LIN {X 0,Y 433.476,Z 320.375,A -85,B 0,C 180,E1 -9833.026,E2 -9833.026} C_VEL
LIN {X 0,Y 436.058,Z 247.757,A -85,B 0,C 180,E1 -9834.679,E2 -9834.679} C_VEL
LIN {X 0,Y 438.537,Z 191.694,A -85,B 0,C 180,E1 -9836.045,E2 -9836.045} C_VEL
LIN {X 0,Y 435.909,Z 167.114,A -85,B 0,C 180,E1 -9837.032,E2 -9837.032} C_VEL
LIN {X 0,Y 432.859,Z 145.77,A -85,B 0,C 180,E1 -9838.059,E2 -9838.059} C_VEL
LIN {X 0,Y 426.886,Z 123.826,A -85,B 0,C 180,E1 -9841.119,E2 -9841.119} C_VEL
LIN {X 0,Y 425.305,Z 118.134,A -85,B 0,C 180,E1 -9841.978,E2 -9841.978} C_VEL
LIN {X 0,Y 425.294,Z 118.133,A -85,B 0,C 180,E1 -9845.337,E2 -9845.337} C_VEL
LIN {X 0,Y 425.279,Z 118.135,A -85,B 0,C 180,E1 -9848.901,E2 -9848.901} C_VEL
LIN {X 0,Y 425.255,Z 118.138,A -85,B 0,C 180,E1 -9852.656,E2 -9852.656} C_VEL
LIN {X 0,Y 425.284,Z 118.131,A -85,B 0,C 180,E1 -9855.283,E2 -9855.283} C_VEL
LIN {X 0,Y 425.247,Z 118.139,A -85,B 0,C 180,E1 -9858.618,E2 -9858.618} C_VEL
LIN {X 0,Y 425.279,Z 118.135,A -85,B 0,C 180,E1 -9861.1,E2 -9861.1} C_VEL
LIN {X 0,Y 425.294,Z 118.135,A -85,B 0,C 180,E1 -9864.664,E2 -9864.664} C_VEL
LIN {X 0,Y 425.262,Z 118.139,A -85,B 0,C 180,E1 -9868.073,E2 -9868.073} C_VEL
LIN {X 0,Y 425.304,Z 118.332,A -85,B 0,C 180,E1 -9870.341,E2 -9870.341} C_VEL
LIN {X 0,Y 427.302,Z 123.447,A -85,B 0,C 180,E1 -9871.42,E2 -9871.42} C_VEL
LIN {X 0,Y 432.761,Z 132.504,A -85,B 0,C 180,E1 -9872.386,E2 -9872.386} C_VEL
LIN {X 0,Y 437.753,Z 142.034,A -85,B 0,C 180,E1 -9873.231,E2 -9873.231} C_VEL
LIN {X 0,Y 440.603,Z 148.513,A -85,B 0,C 180,E1 -9873.713,E2 -9873.713} C_VEL
LIN {X 0,Y 436.849,Z 227.027,A -85,B 0,C 180,E1 -9875.622,E2 -9875.622} C_VEL
LIN {X 0,Y 434.621,Z 288.231,A -85,B 0,C 180,E1 -9877.039,E2 -9877.039} C_VEL
LIN {X 0,Y 433.965,Z 303.14,A -85,B 0,C 180,E1 -9877.553,E2 -9877.553} C_VEL
LIN {X 0,Y 433.141,Z 318.479,A -85,B 0,C 180,E1 -9878.276,E2 -9878.276} C_VEL
LIN {X 0,Y 432.336,Z 331.205,A -85,B 0,C 180,E1 -9879.046,E2 -9879.046} C_VEL
LIN {X 0,Y 431.344,Z 344.128,A -85,B 0,C 180,E1 -9879.992,E2 -9879.992} C_VEL
LIN {X 0,Y 430.278,Z 357.22,A -85,B 0,C 180,E1 -9881.159,E2 -9881.159} C_VEL
LIN {X 0,Y 429.205,Z 368.572,A -85,B 0,C 180,E1 -9882.367,E2 -9882.367} C_VEL
LIN {X 0,Y 428.183,Z 379.818,A -85,B 0,C 180,E1 -9883.798,E2 -9883.798} C_VEL
LIN {X 0,Y 427.387,Z 389.291,A -85,B 0,C 180,E1 -9885.234,E2 -9885.234} C_VEL
LIN {X 0,Y 426.432,Z 398.569,A -85,B 0,C 180,E1 -9886.903,E2 -9886.903} C_VEL
LIN {X 0,Y 425.775,Z 406.243,A -85,B 0,C 180,E1 -9888.576,E2 -9888.576} C_VEL
LIN {X 0,Y 425.268,Z 413.343,A -85,B 0,C 180,E1 -9890.488,E2 -9890.488} C_VEL
LIN {X 0,Y 424.809,Z 418.9,A -85,B 0,C 180,E1 -9892.395,E2 -9892.395} C_VEL
LIN {X 0,Y 424.497,Z 423.037,A -85,B 0,C 180,E1 -9894.299,E2 -9894.299} C_VEL
LIN {X 0,Y 424.444,Z 425.857,A -85,B 0,C 180,E1 -9896.203,E2 -9896.203} C_VEL
LIN {X 0,Y 424.285,Z 427.454,A -85,B 0,C 180,E1 -9898.102,E2 -9898.102} C_VEL
LIN {X 0,Y 424.198,Z 427.83,A -85,B 0,C 180,E1 -9900,E2 -9900} C_VEL
LIN {X 0,Y 424.232,Z 426.986,A -85,B 0,C 180,E1 -9901.899,E2 -9901.899} C_VEL
LIN {X 0,Y 424.347,Z 424.903,A -85,B 0,C 180,E1 -9903.799,E2 -9903.799} C_VEL
LIN {X 0,Y 424.456,Z 421.542,A -85,B 0,C 180,E1 -9905.702,E2 -9905.702} C_VEL
LIN {X 0,Y 424.638,Z 416.847,A -85,B 0,C 180,E1 -9907.609,E2 -9907.609} C_VEL
LIN {X 0,Y 424.941,Z 410.703,A -85,B 0,C 180,E1 -9909.52,E2 -9909.52} C_VEL
LIN {X 0,Y 425.467,Z 402.93,A -85,B 0,C 180,E1 -9911.433,E2 -9911.433} C_VEL
LIN {X 0,Y 425.898,Z 394.118,A -85,B 0,C 180,E1 -9913.196,E2 -9913.196} C_VEL
LIN {X 0,Y 426.684,Z 384.46,A -85,B 0,C 180,E1 -9914.792,E2 -9914.792} C_VEL
LIN {X 0,Y 427.452,Z 374.109,A -85,B 0,C 180,E1 -9916.231,E2 -9916.231} C_VEL
LIN {X 0,Y 428.404,Z 361.628,A -85,B 0,C 180,E1 -9917.678,E2 -9917.678} C_VEL
LIN {X 0,Y 429.284,Z 349.36,A -85,B 0,C 180,E1 -9918.865,E2 -9918.865} C_VEL
LIN {X 0,Y 430.123,Z 335.923,A -85,B 0,C 180,E1 -9919.944,E2 -9919.944} C_VEL
LIN {X 0,Y 431.021,Z 321.131,A -85,B 0,C 180,E1 -9920.897,E2 -9920.897} C_VEL
LIN {X 0,Y 431.726,Z 306.43,A -85,B 0,C 180,E1 -9921.642,E2 -9921.642} C_VEL
LIN {X 0,Y 432.318,Z 290.546,A -85,B 0,C 180,E1 -9922.239,E2 -9922.239} C_VEL
LIN {X 0,Y 432.751,Z 273.967,A -85,B 0,C 180,E1 -9922.656,E2 -9922.656} C_VEL
LIN {X 0,Y 435.763,Z 148.938,A -85,B 0,C 180,E1 -9925.144,E2 -9925.144} C_VEL
LIN {X 0,Y 435.826,Z 144.558,A -85,B 0,C 180,E1 -9925.236,E2 -9925.236} C_VEL
LIN {X 0,Y 427.552,Z 123.717,A -85,B 0,C 180,E1 -9926.145,E2 -9926.145} C_VEL
LIN {X 0,Y 425.381,Z 118.566,A -85,B 0,C 180,E1 -9926.383,E2 -9926.383} C_VEL
LIN {X 0,Y 425.309,Z 118.131,A -85,B 0,C 180,E1 -9926.44,E2 -9926.44} C_VEL
LIN {X 0,Y 425.285,Z 118.138,A -85,B 0,C 180,E1 -9929.72,E2 -9929.72} C_VEL
LIN {X 0,Y 425.271,Z 118.136,A -85,B 0,C 180,E1 -9933.049,E2 -9933.049} C_VEL
LIN {X 0,Y 425.282,Z 118.135,A -85,B 0,C 180,E1 -9935.928,E2 -9935.928} C_VEL
LIN {X 0,Y 425.264,Z 118.137,A -85,B 0,C 180,E1 -9939.038,E2 -9939.038} C_VEL
LIN {X 0,Y 425.259,Z 118.135,A -85,B 0,C 180,E1 -9942.656,E2 -9942.656} C_VEL
LIN {X 0,Y 425.287,Z 118.121,A -85,B 0,C 180,E1 -9945.283,E2 -9945.283} C_VEL
LIN {X 0,Y 425.251,Z 118.129,A -85,B 0,C 180,E1 -9948.619,E2 -9948.619} C_VEL
LIN {X 0,Y 425.286,Z 118.138,A -85,B 0,C 180,E1 -9951.1,E2 -9951.1} C_VEL
LIN {X 0,Y 425.297,Z 118.117,A -85,B 0,C 180,E1 -9954.664,E2 -9954.664} C_VEL
LIN {X 0,Y 425.263,Z 118.135,A -85,B 0,C 180,E1 -9958.073,E2 -9958.073} C_VEL
LIN {X 0,Y 425.307,Z 118.126,A -85,B 0,C 180,E1 -9961.366,E2 -9961.366} C_VEL
LIN {X 0,Y 425.263,Z 118.137,A -85,B 0,C 180,E1 -9964.553,E2 -9964.553} C_VEL
LIN {X 0,Y 425.294,Z 118.131,A -85,B 0,C 180,E1 -9967.73,E2 -9967.73} C_VEL
LIN {X 0,Y 425.363,Z 118.121,A -85,B 0,C 180,E1 -9970.704,E2 -9970.704} C_VEL
LIN {X 0,Y 425.326,Z 118.123,A -85,B 0,C 180,E1 -9973.686,E2 -9973.686} C_VEL
LIN {X 0,Y 425.397,Z 118.118,A -85,B 0,C 180,E1 -9977.097,E2 -9977.097} C_VEL
LIN {X 0,Y 425.391,Z 118.118,A -85,B 0,C 180,E1 -9977.809,E2 -9977.809} C_VEL
LIN {X 0,Y 424.671,Z 118.212,A -85,B 0,C 180,E1 -9978.599,E2 -9978.599} C_VEL
LIN {X 0,Y 421.798,Z 118.565,A -85,B 0,C 180,E1 -9979.883,E2 -9979.883} C_VEL
LIN {X 0,Y 419.433,Z 118.863,A -85,B 0,C 180,E1 -9980.92,E2 -9980.92} C_VEL
LIN {X 0,Y 418.468,Z 118.982,A -85,B 0,C 180,E1 -9981.721,E2 -9981.721} C_VEL
LIN {X 0,Y 418.414,Z 118.988,A -85,B 0,C 180,E1 -9981.992,E2 -9981.992} C_VEL
LIN {X 0,Y 418.469,Z 118.985,A -85,B 0,C 180,E1 -9984.217,E2 -9984.217} C_VEL
LIN {X 0,Y 418.285,Z 119.156,A -85,B 0,C 180,E1 -9986.177,E2 -9986.177} C_VEL
LIN {X 0,Y 420.692,Z 127.345,A -85,B 0,C 180,E1 -9987.606,E2 -9987.606} C_VEL
LIN {X 0,Y 424.262,Z 143.272,A -85,B 0,C 180,E1 -9990.245,E2 -9990.245} C_VEL
LIN {X 0,Y 427.065,Z 154.574,A -85,B 0,C 180,E1 -9990.638,E2 -9990.638} C_VEL
LIN {X 0,Y 430.401,Z 170.837,A -85,B 0,C 180,E1 -9991.151,E2 -9991.151} C_VEL
LIN {X 0,Y 427.922,Z 309.723,A -85,B 0,C 180,E1 -9993.56,E2 -9993.56} C_VEL
LIN {X 0,Y 427.342,Z 325.024,A -85,B 0,C 180,E1 -9994.008,E2 -9994.008} C_VEL
LIN {X 0,Y 426.606,Z 339.301,A -85,B 0,C 180,E1 -9994.606,E2 -9994.606} C_VEL
LIN {X 0,Y 425.719,Z 352.541,A -85,B 0,C 180,E1 -9995.328,E2 -9995.328} C_VEL
LIN {X 0,Y 424.65,Z 366.851,A -85,B 0,C 180,E1 -9996.323,E2 -9996.323} C_VEL
LIN {X 0,Y 423.516,Z 379.354,A -85,B 0,C 180,E1 -9997.389,E2 -9997.389} C_VEL
LIN {X 0,Y 422.318,Z 392.27,A -85,B 0,C 180,E1 -9998.734,E2 -9998.734} C_VEL
LIN {X 0,Y 421.206,Z 403.348,A -85,B 0,C 180,E1 -10000.118,E2 -10000.118} C_VEL
LIN {X 0,Y 420.207,Z 413.193,A -85,B 0,C 180,E1 -10001.578,E2 -10001.578} C_VEL
LIN {X 0,Y 419.231,Z 423.087,A -85,B 0,C 180,E1 -10003.344,E2 -10003.344} C_VEL
LIN {X 0,Y 418.471,Z 431.173,A -85,B 0,C 180,E1 -10005.089,E2 -10005.089} C_VEL
LIN {X 0,Y 417.884,Z 438.749,A -85,B 0,C 180,E1 -10007.117,E2 -10007.117} C_VEL
LIN {X 0,Y 417.436,Z 444.47,A -85,B 0,C 180,E1 -10009.055,E2 -10009.055} C_VEL
LIN {X 0,Y 417.228,Z 448.297,A -85,B 0,C 180,E1 -10010.716,E2 -10010.716} C_VEL
LIN {X 0,Y 416.957,Z 451.799,A -85,B 0,C 180,E1 -10012.81,E2 -10012.81} C_VEL
LIN {X 0,Y 416.84,Z 453.914,A -85,B 0,C 180,E1 -10014.93,E2 -10014.93} C_VEL
LIN {X 0,Y 416.81,Z 454.647,A -85,B 0,C 180,E1 -10017.082,E2 -10017.082} C_VEL
LIN {X 0,Y 416.88,Z 453.936,A -85,B 0,C 180,E1 -10019.268,E2 -10019.268} C_VEL
LIN {X 0,Y 416.959,Z 452.622,A -85,B 0,C 180,E1 -10020.725,E2 -10020.725} C_VEL
LIN {X 0,Y 417.123,Z 449.953,A -85,B 0,C 180,E1 -10022.626,E2 -10022.626} C_VEL
LIN {X 0,Y 417.374,Z 446.422,A -85,B 0,C 180,E1 -10024.401,E2 -10024.401} C_VEL
LIN {X 0,Y 417.655,Z 441.894,A -85,B 0,C 180,E1 -10026.127,E2 -10026.127} C_VEL
LIN {X 0,Y 418.184,Z 435.407,A -85,B 0,C 180,E1 -10028.086,E2 -10028.086} C_VEL
LIN {X 0,Y 418.9,Z 427.843,A -85,B 0,C 180,E1 -10029.921,E2 -10029.921} C_VEL
LIN {X 0,Y 419.836,Z 418.621,A -85,B 0,C 180,E1 -10031.754,E2 -10031.754} C_VEL
LIN {X 0,Y 420.792,Z 409.737,A -85,B 0,C 180,E1 -10033.218,E2 -10033.218} C_VEL
LIN {X 0,Y 421.901,Z 398.872,A -85,B 0,C 180,E1 -10034.733,E2 -10034.733} C_VEL
LIN {X 0,Y 423.054,Z 387.69,A -85,B 0,C 180,E1 -10036.035,E2 -10036.035} C_VEL
LIN {X 0,Y 424.244,Z 375.52,A -85,B 0,C 180,E1 -10037.218,E2 -10037.218} C_VEL
LIN {X 0,Y 425.412,Z 362.05,A -85,B 0,C 180,E1 -10038.296,E2 -10038.296} C_VEL
LIN {X 0,Y 426.457,Z 348.268,A -85,B 0,C 180,E1 -10039.182,E2 -10039.182} C_VEL
LIN {X 0,Y 427.423,Z 333.071,A -85,B 0,C 180,E1 -10039.937,E2 -10039.937} C_VEL
LIN {X 0,Y 428.11,Z 318.612,A -85,B 0,C 180,E1 -10040.459,E2 -10040.459} C_VEL
LIN {X 0,Y 428.609,Z 302.995,A -85,B 0,C 180,E1 -10040.831,E2 -10040.831} C_VEL
LIN {X 0,Y 431.166,Z 166.127,A -85,B 0,C 180,E1 -10043.203,E2 -10043.203} C_VEL
LIN {X 0,Y 427.935,Z 148.87,A -85,B 0,C 180,E1 -10043.755,E2 -10043.755} C_VEL
LIN {X 0,Y 424.959,Z 141.623,A -85,B 0,C 180,E1 -10044.132,E2 -10044.132} C_VEL
LIN {X 0,Y 421.22,Z 128.241,A -85,B 0,C 180,E1 -10046.017,E2 -10046.017} C_VEL
LIN {X 0,Y 418.253,Z 119.013,A -85,B 0,C 180,E1 -10047.386,E2 -10047.386} C_VEL
LIN {X 0,Y 418.271,Z 119.005,A -85,B 0,C 180,E1 -10050.895,E2 -10050.895} C_VEL
LIN {X 0,Y 418.343,Z 119.17,A -85,B 0,C 180,E1 -10053.285,E2 -10053.285} C_VEL
LIN {X 0,Y 420.465,Z 124.425,A -85,B 0,C 180,E1 -10053.527,E2 -10053.527} C_VEL
LIN {X 0,Y 428.257,Z 143.1,A -85,B 0,C 180,E1 -10054.384,E2 -10054.384} C_VEL
LIN {X 0,Y 429.352,Z 145.894,A -85,B 0,C 180,E1 -10054.505,E2 -10054.505} C_VEL
LIN {X 0,Y 425.813,Z 284.514,A -85,B 0,C 180,E1 -10057.37,E2 -10057.37} C_VEL
LIN {X 0,Y 425.291,Z 300.109,A -85,B 0,C 180,E1 -10057.884,E2 -10057.884} C_VEL
LIN {X 0,Y 424.58,Z 315.42,A -85,B 0,C 180,E1 -10058.585,E2 -10058.585} C_VEL
LIN {X 0,Y 423.681,Z 330.521,A -85,B 0,C 180,E1 -10059.487,E2 -10059.487} C_VEL
LIN {X 0,Y 422.828,Z 343.594,A -85,B 0,C 180,E1 -10060.457,E2 -10060.457} C_VEL
LIN {X 0,Y 421.904,Z 356.853,A -85,B 0,C 180,E1 -10061.655,E2 -10061.655} C_VEL
LIN {X 0,Y 420.946,Z 369.299,A -85,B 0,C 180,E1 -10063.011,E2 -10063.011} C_VEL
LIN {X 0,Y 420.094,Z 380.508,A -85,B 0,C 180,E1 -10064.474,E2 -10064.474} C_VEL
LIN {X 0,Y 419.355,Z 389.987,A -85,B 0,C 180,E1 -10065.936,E2 -10065.936} C_VEL
LIN {X 0,Y 418.741,Z 399.242,A -85,B 0,C 180,E1 -10067.643,E2 -10067.643} C_VEL
LIN {X 0,Y 418.126,Z 406.928,A -85,B 0,C 180,E1 -10069.345,E2 -10069.345} C_VEL
LIN {X 0,Y 417.739,Z 414.027,A -85,B 0,C 180,E1 -10071.291,E2 -10071.291} C_VEL
LIN {X 0,Y 417.441,Z 419.577,A -85,B 0,C 180,E1 -10073.232,E2 -10073.232} C_VEL
LIN {X 0,Y 417.253,Z 423.717,A -85,B 0,C 180,E1 -10075.169,E2 -10075.169} C_VEL
LIN {X 0,Y 417.274,Z 426.53,A -85,B 0,C 180,E1 -10077.103,E2 -10077.103} C_VEL
LIN {X 0,Y 417.116,Z 428.105,A -85,B 0,C 180,E1 -10079.034,E2 -10079.034} C_VEL
LIN {X 0,Y 417.159,Z 428.456,A -85,B 0,C 180,E1 -10080.965,E2 -10080.965} C_VEL
LIN {X 0,Y 417.307,Z 427.591,A -85,B 0,C 180,E1 -10082.896,E2 -10082.896} C_VEL
LIN {X 0,Y 417.35,Z 425.512,A -85,B 0,C 180,E1 -10084.83,E2 -10084.83} C_VEL
LIN {X 0,Y 417.706,Z 421.785,A -85,B 0,C 180,E1 -10086.933,E2 -10086.933} C_VEL
LIN {X 0,Y 418.018,Z 417.459,A -85,B 0,C 180,E1 -10088.703,E2 -10088.703} C_VEL
LIN {X 0,Y 418.538,Z 411.293,A -85,B 0,C 180,E1 -10090.644,E2 -10090.644} C_VEL
LIN {X 0,Y 419.232,Z 403.488,A -85,B 0,C 180,E1 -10092.587,E2 -10092.587} C_VEL
LIN {X 0,Y 420.006,Z 395.644,A -85,B 0,C 180,E1 -10094.189,E2 -10094.189} C_VEL
LIN {X 0,Y 420.973,Z 386.577,A -85,B 0,C 180,E1 -10095.741,E2 -10095.741} C_VEL
LIN {X 0,Y 421.96,Z 376.468,A -85,B 0,C 180,E1 -10097.195,E2 -10097.195} C_VEL
LIN {X 0,Y 423.082,Z 364.868,A -85,B 0,C 180,E1 -10098.601,E2 -10098.601} C_VEL
LIN {X 0,Y 424.377,Z 351.134,A -85,B 0,C 180,E1 -10099.972,E2 -10099.972} C_VEL
LIN {X 0,Y 425.556,Z 337.924,A -85,B 0,C 180,E1 -10101.051,E2 -10101.051} C_VEL
LIN {X 0,Y 426.562,Z 323.478,A -85,B 0,C 180,E1 -10102.013,E2 -10102.013} C_VEL
LIN {X 0,Y 427.571,Z 308.227,A -85,B 0,C 180,E1 -10102.802,E2 -10102.802} C_VEL
LIN {X 0,Y 428.387,Z 292.392,A -85,B 0,C 180,E1 -10103.411,E2 -10103.411} C_VEL
LIN {X 0,Y 429.03,Z 274.518,A -85,B 0,C 180,E1 -10103.886,E2 -10103.886} C_VEL
LIN {X 0,Y 432.057,Z 206.122,A -85,B 0,C 180,E1 -10105.535,E2 -10105.535} C_VEL
LIN {X 0,Y 435.05,Z 152.54,A -85,B 0,C 180,E1 -10106.899,E2 -10106.899} C_VEL
LIN {X 0,Y 429.528,Z 141.704,A -85,B 0,C 180,E1 -10107.869,E2 -10107.869} C_VEL
LIN {X 0,Y 423.452,Z 131.573,A -85,B 0,C 180,E1 -10108.995,E2 -10108.995} C_VEL
LIN {X 0,Y 421.069,Z 127.829,A -85,B 0,C 180,E1 -10109.498,E2 -10109.498} C_VEL
LIN {X 0,Y 419.163,Z 121.743,A -85,B 0,C 180,E1 -10111.88,E2 -10111.88} C_VEL
LIN {X 0,Y 418.224,Z 119.016,A -85,B 0,C 180,E1 -10113.214,E2 -10113.214} C_VEL
LIN {X 0,Y 418.243,Z 119.013,A -85,B 0,C 180,E1 -10116.237,E2 -10116.237} C_VEL
LIN {X 0,Y 418.199,Z 119.02,A -85,B 0,C 180,E1 -10119.688,E2 -10119.688} C_VEL
LIN {X 0,Y 418.207,Z 119.018,A -85,B 0,C 180,E1 -10122.318,E2 -10122.318} C_VEL
LIN {X 0,Y 418.234,Z 119.014,A -85,B 0,C 180,E1 -10125.108,E2 -10125.108} C_VEL
LIN {X 0,Y 418.218,Z 119.017,A -85,B 0,C 180,E1 -10127.764,E2 -10127.764} C_VEL
LIN {X 0,Y 418.264,Z 119.189,A -85,B 0,C 180,E1 -10131.251,E2 -10131.251} C_VEL
LIN {X 0,Y 420.236,Z 124.674,A -85,B 0,C 180,E1 -10133.393,E2 -10133.393} C_VEL
LIN {X 0,Y 422.812,Z 132.475,A -85,B 0,C 180,E1 -10135.857,E2 -10135.857} C_VEL
LIN {X 0,Y 425.058,Z 140.837,A -85,B 0,C 180,E1 -10138.056,E2 -10138.056} C_VEL
LIN {X 0,Y 427.012,Z 150.076,A -85,B 0,C 180,E1 -10140.141,E2 -10140.141} C_VEL
LIN {X 0,Y 426.311,Z 155.998,A -85,B 0,C 180,E1 -10141.195,E2 -10141.195} C_VEL
LIN {X 0,Y 429.906,Z 173.135,A -85,B 0,C 180,E1 -10142.192,E2 -10142.192} C_VEL
LIN {X 0,Y 432.21,Z 187.065,A -85,B 0,C 180,E1 -10142.874,E2 -10142.874} C_VEL
LIN {X 0,Y 433.425,Z 198.784,A -85,B 0,C 180,E1 -10143.353,E2 -10143.353} C_VEL
LIN {X 0,Y 429.495,Z 281.182,A -85,B 0,C 180,E1 -10145.37,E2 -10145.37} C_VEL
LIN {X 0,Y 427.704,Z 328.281,A -85,B 0,C 180,E1 -10146.485,E2 -10146.485} C_VEL
LIN {X 0,Y 426.584,Z 344.904,A -85,B 0,C 180,E1 -10147.062,E2 -10147.062} C_VEL
LIN {X 0,Y 425.045,Z 368.196,A -85,B 0,C 180,E1 -10148.155,E2 -10148.155} C_VEL
LIN {X 0,Y 424.013,Z 381.982,A -85,B 0,C 180,E1 -10148.996,E2 -10148.996} C_VEL
LIN {X 0,Y 423.04,Z 394.637,A -85,B 0,C 180,E1 -10149.962,E2 -10149.962} C_VEL
LIN {X 0,Y 421.807,Z 407.625,A -85,B 0,C 180,E1 -10151.166,E2 -10151.166} C_VEL
LIN {X 0,Y 420.765,Z 419.459,A -85,B 0,C 180,E1 -10152.503,E2 -10152.503} C_VEL
LIN {X 0,Y 419.746,Z 430.266,A -85,B 0,C 180,E1 -10153.962,E2 -10153.962} C_VEL
LIN {X 0,Y 418.815,Z 440.763,A -85,B 0,C 180,E1 -10155.669,E2 -10155.669} C_VEL
LIN {X 0,Y 418.115,Z 449.456,A -85,B 0,C 180,E1 -10157.378,E2 -10157.378} C_VEL
LIN {X 0,Y 417.766,Z 455.753,A -85,B 0,C 180,E1 -10158.845,E2 -10158.845} C_VEL
LIN {X 0,Y 417.329,Z 462.608,A -85,B 0,C 180,E1 -10160.794,E2 -10160.794} C_VEL
LIN {X 0,Y 417.183,Z 467.962,A -85,B 0,C 180,E1 -10162.741,E2 -10162.741} C_VEL
LIN {X 0,Y 417.089,Z 471.027,A -85,B 0,C 180,E1 -10164.197,E2 -10164.197} C_VEL
LIN {X 0,Y 417.015,Z 474.038,A -85,B 0,C 180,E1 -10166.135,E2 -10166.135} C_VEL
LIN {X 0,Y 417.107,Z 475.831,A -85,B 0,C 180,E1 -10168.069,E2 -10168.069} C_VEL
LIN {X 0,Y 417.008,Z 476.43,A -85,B 0,C 180,E1 -10170,E2 -10170} C_VEL
LIN {X 0,Y 417.105,Z 475.816,A -85,B 0,C 180,E1 -10171.931,E2 -10171.931} C_VEL
LIN {X 0,Y 417.022,Z 473.988,A -85,B 0,C 180,E1 -10173.865,E2 -10173.865} C_VEL
LIN {X 0,Y 417.103,Z 470.93,A -85,B 0,C 180,E1 -10175.802,E2 -10175.802} C_VEL
LIN {X 0,Y 417.213,Z 466.566,A -85,B 0,C 180,E1 -10177.745,E2 -10177.745} C_VEL
LIN {X 0,Y 417.373,Z 460.79,A -85,B 0,C 180,E1 -10179.694,E2 -10179.694} C_VEL
LIN {X 0,Y 417.826,Z 453.441,A -85,B 0,C 180,E1 -10181.645,E2 -10181.645} C_VEL
LIN {X 0,Y 418.352,Z 445.454,A -85,B 0,C 180,E1 -10183.367,E2 -10183.367} C_VEL
LIN {X 0,Y 419.132,Z 435.942,A -85,B 0,C 180,E1 -10185.064,E2 -10185.064} C_VEL
LIN {X 0,Y 420.01,Z 426.133,A -85,B 0,C 180,E1 -10186.527,E2 -10186.527} C_VEL
LIN {X 0,Y 420.865,Z 415.606,A -85,B 0,C 180,E1 -10187.855,E2 -10187.855} C_VEL
LIN {X 0,Y 421.863,Z 403.993,A -85,B 0,C 180,E1 -10189.083,E2 -10189.083} C_VEL
LIN {X 0,Y 422.961,Z 391.607,A -85,B 0,C 180,E1 -10190.169,E2 -10190.169} C_VEL
LIN {X 0,Y 423.984,Z 378.111,A -85,B 0,C 180,E1 -10191.133,E2 -10191.133} C_VEL
LIN {X 0,Y 425.004,Z 363.864,A -85,B 0,C 180,E1 -10191.929,E2 -10191.929} C_VEL
LIN {X 0,Y 425.699,Z 349.61,A -85,B 0,C 180,E1 -10192.54,E2 -10192.54} C_VEL
LIN {X 0,Y 426.927,Z 326.53,A -85,B 0,C 180,E1 -10193.303,E2 -10193.303} C_VEL
LIN {X 0,Y 430.632,Z 235.57,A -85,B 0,C 180,E1 -10195.466,E2 -10195.466} C_VEL
LIN {X 0,Y 432.676,Z 192.835,A -85,B 0,C 180,E1 -10196.555,E2 -10196.555} C_VEL
LIN {X 0,Y 430.315,Z 169.02,A -85,B 0,C 180,E1 -10197.549,E2 -10197.549} C_VEL
LIN {X 0,Y 427.476,Z 148.909,A -85,B 0,C 180,E1 -10198.546,E2 -10198.546} C_VEL
LIN {X 0,Y 423.411,Z 137.794,A -85,B 0,C 180,E1 -10199.581,E2 -10199.581} C_VEL
LIN {X 0,Y 418.279,Z 119.007,A -85,B 0,C 180,E1 -10202.311,E2 -10202.311} C_VEL
LIN {X 0,Y 418.249,Z 119.013,A -85,B 0,C 180,E1 -10204.842,E2 -10204.842} C_VEL
LIN {X 0,Y 418.237,Z 119.012,A -85,B 0,C 180,E1 -10208.444,E2 -10208.444} C_VEL
LIN {X 0,Y 418.218,Z 119.012,A -85,B 0,C 180,E1 -10212.236,E2 -10212.236} C_VEL
LIN {X 0,Y 418.234,Z 119.01,A -85,B 0,C 180,E1 -10215.109,E2 -10215.109} C_VEL
LIN {X 0,Y 418.218,Z 119.012,A -85,B 0,C 180,E1 -10217.764,E2 -10217.764} C_VEL
LIN {X 0,Y 418.237,Z 119.014,A -85,B 0,C 180,E1 -10221.557,E2 -10221.557} C_VEL
LIN {X 0,Y 418.25,Z 119.012,A -85,B 0,C 180,E1 -10225.158,E2 -10225.158} C_VEL
LIN {X 0,Y 418.243,Z 119.013,A -85,B 0,C 180,E1 -10227.472,E2 -10227.472} C_VEL
LIN {X 0,Y 418.275,Z 119.133,A -85,B 0,C 180,E1 -10229.366,E2 -10229.366} C_VEL
LIN {X 0,Y 418.771,Z 120.997,A -85,B 0,C 180,E1 -10229.77,E2 -10229.77} C_VEL
LIN {X 0,Y 420.148,Z 123.987,A -85,B 0,C 180,E1 -10230.487,E2 -10230.487} C_VEL
LIN {X 0,Y 426.123,Z 133.617,A -85,B 0,C 180,E1 -10231.643,E2 -10231.643} C_VEL
LIN {X 0,Y 430.993,Z 142.386,A -85,B 0,C 180,E1 -10232.52,E2 -10232.52} C_VEL
LIN {X 0,Y 434.88,Z 150.985,A -85,B 0,C 180,E1 -10233.217,E2 -10233.217} C_VEL
LIN {X 0,Y 430.518,Z 234.6,A -85,B 0,C 180,E1 -10235.304,E2 -10235.304} C_VEL
LIN {X 0,Y 428.335,Z 289.381,A -85,B 0,C 180,E1 -10236.618,E2 -10236.618} C_VEL
LIN {X 0,Y 427.588,Z 305.204,A -85,B 0,C 180,E1 -10237.19,E2 -10237.19} C_VEL
LIN {X 0,Y 426.693,Z 320.173,A -85,B 0,C 180,E1 -10237.93,E2 -10237.93} C_VEL
LIN {X 0,Y 425.713,Z 334.367,A -85,B 0,C 180,E1 -10238.831,E2 -10238.831} C_VEL
LIN {X 0,Y 424.548,Z 348.176,A -85,B 0,C 180,E1 -10239.91,E2 -10239.91} C_VEL
LIN {X 0,Y 423.39,Z 360.836,A -85,B 0,C 180,E1 -10241.114,E2 -10241.114} C_VEL
LIN {X 0,Y 422.308,Z 371.547,A -85,B 0,C 180,E1 -10242.319,E2 -10242.319} C_VEL
LIN {X 0,Y 421.288,Z 382.377,A -85,B 0,C 180,E1 -10243.774,E2 -10243.774} C_VEL
LIN {X 0,Y 420.398,Z 391.524,A -85,B 0,C 180,E1 -10245.23,E2 -10245.23} C_VEL
LIN {X 0,Y 419.431,Z 400.498,A -85,B 0,C 180,E1 -10246.926,E2 -10246.926} C_VEL
LIN {X 0,Y 418.837,Z 406.906,A -85,B 0,C 180,E1 -10248.384,E2 -10248.384} C_VEL
LIN {X 0,Y 418.279,Z 413.962,A -85,B 0,C 180,E1 -10250.327,E2 -10250.327} C_VEL
LIN {X 0,Y 417.792,Z 419.473,A -85,B 0,C 180,E1 -10252.266,E2 -10252.266} C_VEL
LIN {X 0,Y 417.455,Z 423.565,A -85,B 0,C 180,E1 -10254.203,E2 -10254.203} C_VEL
LIN {X 0,Y 417.384,Z 426.346,A -85,B 0,C 180,E1 -10256.138,E2 -10256.138} C_VEL
LIN {X 0,Y 417.208,Z 427.896,A -85,B 0,C 180,E1 -10258.07,E2 -10258.07} C_VEL
LIN {X 0,Y 417.112,Z 428.222,A -85,B 0,C 180,E1 -10260,E2 -10260} C_VEL
LIN {X 0,Y 417.157,Z 427.324,A -85,B 0,C 180,E1 -10261.931,E2 -10261.931} C_VEL
LIN {X 0,Y 417.252,Z 425.193,A -85,B 0,C 180,E1 -10263.863,E2 -10263.863} C_VEL
LIN {X 0,Y 417.383,Z 421.774,A -85,B 0,C 180,E1 -10265.799,E2 -10265.799} C_VEL
LIN {X 0,Y 417.574,Z 417.004,A -85,B 0,C 180,E1 -10267.738,E2 -10267.738} C_VEL
LIN {X 0,Y 417.882,Z 410.774,A -85,B 0,C 180,E1 -10269.682,E2 -10269.682} C_VEL
LIN {X 0,Y 418.355,Z 403.949,A -85,B 0,C 180,E1 -10271.385,E2 -10271.385} C_VEL
LIN {X 0,Y 418.738,Z 396.907,A -85,B 0,C 180,E1 -10272.858,E2 -10272.858} C_VEL
LIN {X 0,Y 419.503,Z 387.256,A -85,B 0,C 180,E1 -10274.555,E2 -10274.555} C_VEL
LIN {X 0,Y 420.289,Z 377.336,A -85,B 0,C 180,E1 -10276.017,E2 -10276.017} C_VEL
LIN {X 0,Y 421.228,Z 365.533,A -85,B 0,C 180,E1 -10277.477,E2 -10277.477} C_VEL
LIN {X 0,Y 422.124,Z 352.523,A -85,B 0,C 180,E1 -10278.819,E2 -10278.819} C_VEL
LIN {X 0,Y 423.049,Z 339.692,A -85,B 0,C 180,E1 -10279.911,E2 -10279.911} C_VEL
LIN {X 0,Y 423.936,Z 325.787,A -85,B 0,C 180,E1 -10280.881,E2 -10280.881} C_VEL
LIN {X 0,Y 424.746,Z 310.546,A -85,B 0,C 180,E1 -10281.724,E2 -10281.724} C_VEL
LIN {X 0,Y 425.373,Z 295.193,A -85,B 0,C 180,E1 -10282.366,E2 -10282.366} C_VEL
LIN {X 0,Y 425.868,Z 279.661,A -85,B 0,C 180,E1 -10282.819,E2 -10282.819} C_VEL
LIN {X 0,Y 429.149,Z 149.841,A -85,B 0,C 180,E1 -10285.474,E2 -10285.474} C_VEL
LIN {X 0,Y 429.007,Z 145.736,A -85,B 0,C 180,E1 -10285.573,E2 -10285.573} C_VEL
LIN {X 0,Y 421.571,Z 127.049,A -85,B 0,C 180,E1 -10286.402,E2 -10286.402} C_VEL
LIN {X 0,Y 418.336,Z 119.6,A -85,B 0,C 180,E1 -10286.757,E2 -10286.757} C_VEL
LIN {X 0,Y 418.245,Z 119.012,A -85,B 0,C 180,E1 -10286.792,E2 -10286.792} C_VEL
LIN {X 0,Y 418.243,Z 119.012,A -85,B 0,C 180,E1 -10290.273,E2 -10290.273} C_VEL
LIN {X 0,Y 418.234,Z 119.015,A -85,B 0,C 180,E1 -10293.679,E2 -10293.679} C_VEL
LIN {X 0,Y 418.24,Z 119.013,A -85,B 0,C 180,E1 -10297.225,E2 -10297.225} C_VEL
LIN {X 0,Y 418.209,Z 119.015,A -85,B 0,C 180,E1 -10300.867,E2 -10300.867} C_VEL
LIN {X 0,Y 418.205,Z 119.012,A -85,B 0,C 180,E1 -10303.729,E2 -10303.729} C_VEL
LIN {X 0,Y 418.201,Z 118.995,A -85,B 0,C 180,E1 -10306.448,E2 -10306.448} C_VEL
LIN {X 0,Y 418.212,Z 119.011,A -85,B 0,C 180,E1 -10309.133,E2 -10309.133} C_VEL
LIN {X 0,Y 418.241,Z 119.007,A -85,B 0,C 180,E1 -10312.776,E2 -10312.776} C_VEL
LIN {X 0,Y 418.235,Z 119.007,A -85,B 0,C 180,E1 -10316.322,E2 -10316.322} C_VEL
LIN {X 0,Y 418.241,Z 119.002,A -85,B 0,C 180,E1 -10319.728,E2 -10319.728} C_VEL
LIN {X 0,Y 418.224,Z 119.017,A -85,B 0,C 180,E1 -10323.017,E2 -10323.017} C_VEL
LIN {X 0,Y 418.258,Z 118.999,A -85,B 0,C 180,E1 -10326.217,E2 -10326.217} C_VEL
LIN {X 0,Y 418.25,Z 119.005,A -85,B 0,C 180,E1 -10329.337,E2 -10329.337} C_VEL
LIN {X 0,Y 418.259,Z 119.013,A -85,B 0,C 180,E1 -10332.395,E2 -10332.395} C_VEL
LIN {X 0,Y 418.279,Z 119.007,A -85,B 0,C 180,E1 -10335.402,E2 -10335.402} C_VEL
LIN {X 0,Y 418.316,Z 119.007,A -85,B 0,C 180,E1 -10338.369,E2 -10338.369} C_VEL
LIN {X 0,Y 418.414,Z 118.988,A -85,B 0,C 180,E1 -10341.992,E2 -10341.992} C_VEL
LIN {X 0,Y 417.781,Z 119.072,A -85,B 0,C 180,E1 -10342.527,E2 -10342.527} C_VEL
LIN {X 0,Y 414.954,Z 119.422,A -85,B 0,C 180,E1 -10343.364,E2 -10343.364} C_VEL
LIN {X 0,Y 412.046,Z 119.786,A -85,B 0,C 180,E1 -10344.211,E2 -10344.211} C_VEL
LIN {X 0,Y 411.318,Z 119.874,A -85,B 0,C 180,E1 -10344.76,E2 -10344.76} C_VEL
LIN {X 0,Y 411.243,Z 120.098,A -85,B 0,C 180,E1 -10345.774,E2 -10345.774} C_VEL
LIN {X 0,Y 414.2,Z 130.215,A -85,B 0,C 180,E1 -10347.569,E2 -10347.569} C_VEL
LIN {X 0,Y 417.199,Z 143.468,A -85,B 0,C 180,E1 -10349.779,E2 -10349.779} C_VEL
LIN {X 0,Y 419.11,Z 149.054,A -85,B 0,C 180,E1 -10350.015,E2 -10350.015} C_VEL
LIN {X 0,Y 423.908,Z 171.508,A -85,B 0,C 180,E1 -10350.754,E2 -10350.754} C_VEL
LIN {X 0,Y 421.374,Z 309.968,A -85,B 0,C 180,E1 -10353.197,E2 -10353.197} C_VEL
LIN {X 0,Y 420.768,Z 325.254,A -85,B 0,C 180,E1 -10353.651,E2 -10353.651} C_VEL
LIN {X 0,Y 419.996,Z 339.529,A -85,B 0,C 180,E1 -10354.258,E2 -10354.258} C_VEL
LIN {X 0,Y 418.992,Z 353.707,A -85,B 0,C 180,E1 -10355.052,E2 -10355.052} C_VEL
LIN {X 0,Y 418.005,Z 366.432,A -85,B 0,C 180,E1 -10355.948,E2 -10355.948} C_VEL
LIN {X 0,Y 416.7,Z 380.204,A -85,B 0,C 180,E1 -10357.145,E2 -10357.145} C_VEL
LIN {X 0,Y 415.474,Z 393.004,A -85,B 0,C 180,E1 -10358.512,E2 -10358.512} C_VEL
LIN {X 0,Y 414.396,Z 402.934,A -85,B 0,C 180,E1 -10359.764,E2 -10359.764} C_VEL
LIN {X 0,Y 413.338,Z 413.023,A -85,B 0,C 180,E1 -10361.276,E2 -10361.276} C_VEL
LIN {X 0,Y 412.443,Z 421.575,A -85,B 0,C 180,E1 -10362.798,E2 -10362.798} C_VEL
LIN {X 0,Y 411.591,Z 430.017,A -85,B 0,C 180,E1 -10364.588,E2 -10364.588} C_VEL
LIN {X 0,Y 411.009,Z 436.636,A -85,B 0,C 180,E1 -10366.289,E2 -10366.289} C_VEL
LIN {X 0,Y 410.581,Z 441.966,A -85,B 0,C 180,E1 -10367.945,E2 -10367.945} C_VEL
LIN {X 0,Y 410.224,Z 447.252,A -85,B 0,C 180,E1 -10370.038,E2 -10370.038} C_VEL
LIN {X 0,Y 409.936,Z 451.206,A -85,B 0,C 180,E1 -10372.212,E2 -10372.212} C_VEL
LIN {X 0,Y 409.796,Z 453.62,A -85,B 0,C 180,E1 -10374.305,E2 -10374.305} C_VEL
LIN {X 0,Y 409.712,Z 454.737,A -85,B 0,C 180,E1 -10376.487,E2 -10376.487} C_VEL
LIN {X 0,Y 409.754,Z 454.434,A -85,B 0,C 180,E1 -10378.702,E2 -10378.702} C_VEL
LIN {X 0,Y 409.878,Z 452.637,A -85,B 0,C 180,E1 -10380.957,E2 -10380.957} C_VEL
LIN {X 0,Y 410.056,Z 449.892,A -85,B 0,C 180,E1 -10382.878,E2 -10382.878} C_VEL
LIN {X 0,Y 410.347,Z 446.214,A -85,B 0,C 180,E1 -10384.704,E2 -10384.704} C_VEL
LIN {X 0,Y 410.773,Z 440.618,A -85,B 0,C 180,E1 -10386.786,E2 -10386.786} C_VEL
LIN {X 0,Y 411.344,Z 434.323,A -85,B 0,C 180,E1 -10388.629,E2 -10388.629} C_VEL
LIN {X 0,Y 412.037,Z 426.919,A -85,B 0,C 180,E1 -10390.403,E2 -10390.403} C_VEL
LIN {X 0,Y 413.06,Z 417.626,A -85,B 0,C 180,E1 -10392.227,E2 -10392.227} C_VEL
LIN {X 0,Y 414.172,Z 408.105,A -85,B 0,C 180,E1 -10393.784,E2 -10393.784} C_VEL
LIN {X 0,Y 415.339,Z 397.121,A -85,B 0,C 180,E1 -10395.291,E2 -10395.291} C_VEL
LIN {X 0,Y 416.636,Z 384.993,A -85,B 0,C 180,E1 -10396.673,E2 -10396.673} C_VEL
LIN {X 0,Y 417.972,Z 371.929,A -85,B 0,C 180,E1 -10397.897,E2 -10397.897} C_VEL
LIN {X 0,Y 419.132,Z 358.932,A -85,B 0,C 180,E1 -10398.896,E2 -10398.896} C_VEL
LIN {X 0,Y 420.225,Z 344.402,A -85,B 0,C 180,E1 -10399.785,E2 -10399.785} C_VEL
LIN {X 0,Y 421.163,Z 329.225,A -85,B 0,C 180,E1 -10400.488,E2 -10400.488} C_VEL
LIN {X 0,Y 421.827,Z 315.103,A -85,B 0,C 180,E1 -10400.958,E2 -10400.958} C_VEL
LIN {X 0,Y 422.254,Z 297.455,A -85,B 0,C 180,E1 -10401.331,E2 -10401.331} C_VEL
LIN {X 0,Y 424.783,Z 166.685,A -85,B 0,C 180,E1 -10403.636,E2 -10403.636} C_VEL
LIN {X 0,Y 421.932,Z 151.429,A -85,B 0,C 180,E1 -10404.138,E2 -10404.138} C_VEL
LIN {X 0,Y 417.911,Z 141.886,A -85,B 0,C 180,E1 -10404.647,E2 -10404.647} C_VEL
LIN {X 0,Y 414.136,Z 128.828,A -85,B 0,C 180,E1 -10406.529,E2 -10406.529} C_VEL
LIN {X 0,Y 411.174,Z 119.893,A -85,B 0,C 180,E1 -10407.859,E2 -10407.859} C_VEL
LIN {X 0,Y 411.221,Z 119.887,A -85,B 0,C 180,E1 -10411.41,E2 -10411.41} C_VEL
LIN {X 0,Y 411.277,Z 119.882,A -85,B 0,C 180,E1 -10412.881,E2 -10412.881} C_VEL
LIN {X 0,Y 412.965,Z 124.424,A -85,B 0,C 180,E1 -10413.096,E2 -10413.096} C_VEL
LIN {X 0,Y 420.673,Z 142.445,A -85,B 0,C 180,E1 -10413.953,E2 -10413.953} C_VEL
LIN {X 0,Y 422.777,Z 148.152,A -85,B 0,C 180,E1 -10414.199,E2 -10414.199} C_VEL
LIN {X 0,Y 419.045,Z 284.518,A -85,B 0,C 180,E1 -10417.082,E2 -10417.082} C_VEL
LIN {X 0,Y 418.509,Z 300.304,A -85,B 0,C 180,E1 -10417.61,E2 -10417.61} C_VEL
LIN {X 0,Y 417.811,Z 314.865,A -85,B 0,C 180,E1 -10418.28,E2 -10418.28} C_VEL
LIN {X 0,Y 416.942,Z 329.33,A -85,B 0,C 180,E1 -10419.14,E2 -10419.14} C_VEL
LIN {X 0,Y 416.036,Z 342.687,A -85,B 0,C 180,E1 -10420.125,E2 -10420.125} C_VEL
LIN {X 0,Y 415.144,Z 355.124,A -85,B 0,C 180,E1 -10421.237,E2 -10421.237} C_VEL
LIN {X 0,Y 414.197,Z 367.798,A -85,B 0,C 180,E1 -10422.599,E2 -10422.599} C_VEL
LIN {X 0,Y 413.158,Z 380.173,A -85,B 0,C 180,E1 -10424.206,E2 -10424.206} C_VEL
LIN {X 0,Y 412.389,Z 389.783,A -85,B 0,C 180,E1 -10425.693,E2 -10425.693} C_VEL
LIN {X 0,Y 411.737,Z 399.159,A -85,B 0,C 180,E1 -10427.43,E2 -10427.43} C_VEL
LIN {X 0,Y 411.097,Z 406.925,A -85,B 0,C 180,E1 -10429.16,E2 -10429.16} C_VEL
LIN {X 0,Y 410.698,Z 414.136,A -85,B 0,C 180,E1 -10431.14,E2 -10431.14} C_VEL
LIN {X 0,Y 410.381,Z 419.766,A -85,B 0,C 180,E1 -10433.115,E2 -10433.115} C_VEL
LIN {X 0,Y 410.189,Z 423.967,A -85,B 0,C 180,E1 -10435.085,E2 -10435.085} C_VEL
LIN {X 0,Y 410.208,Z 426.842,A -85,B 0,C 180,E1 -10437.053,E2 -10437.053} C_VEL
LIN {X 0,Y 410.035,Z 428.482,A -85,B 0,C 180,E1 -10439.018,E2 -10439.018} C_VEL
LIN {X 0,Y 410.077,Z 428.892,A -85,B 0,C 180,E1 -10440.982,E2 -10440.982} C_VEL
LIN {X 0,Y 410.243,Z 428.078,A -85,B 0,C 180,E1 -10442.946,E2 -10442.946} C_VEL
LIN {X 0,Y 410.343,Z 427.214,A -85,B 0,C 180,E1 -10443.928,E2 -10443.928} C_VEL
LIN {X 0,Y 410.428,Z 424.561,A -85,B 0,C 180,E1 -10445.897,E2 -10445.897} C_VEL
LIN {X 0,Y 410.767,Z 420.595,A -85,B 0,C 180,E1 -10447.867,E2 -10447.867} C_VEL
LIN {X 0,Y 411.337,Z 415.23,A -85,B 0,C 180,E1 -10449.837,E2 -10449.837} C_VEL
LIN {X 0,Y 411.942,Z 408.33,A -85,B 0,C 180,E1 -10451.813,E2 -10451.813} C_VEL
LIN {X 0,Y 412.682,Z 400.898,A -85,B 0,C 180,E1 -10453.54,E2 -10453.54} C_VEL
LIN {X 0,Y 413.754,Z 391.859,A -85,B 0,C 180,E1 -10455.265,E2 -10455.265} C_VEL
LIN {X 0,Y 414.866,Z 380.956,A -85,B 0,C 180,E1 -10456.991,E2 -10456.991} C_VEL
LIN {X 0,Y 416.066,Z 369.74,A -85,B 0,C 180,E1 -10458.464,E2 -10458.464} C_VEL
LIN {X 0,Y 417.341,Z 357.436,A -85,B 0,C 180,E1 -10459.81,E2 -10459.81} C_VEL
LIN {X 0,Y 418.468,Z 345.502,A -85,B 0,C 180,E1 -10460.909,E2 -10460.909} C_VEL
LIN {X 0,Y 419.717,Z 330.912,A -85,B 0,C 180,E1 -10462.003,E2 -10462.003} C_VEL
LIN {X 0,Y 420.734,Z 317.464,A -85,B 0,C 180,E1 -10462.818,E2 -10462.818} C_VEL
LIN {X 0,Y 421.711,Z 302.301,A -85,B 0,C 180,E1 -10463.529,E2 -10463.529} C_VEL
LIN {X 0,Y 422.426,Z 287.203,A -85,B 0,C 180,E1 -10464.054,E2 -10464.054} C_VEL
LIN {X 0,Y 425.929,Z 212.161,A -85,B 0,C 180,E1 -10465.929,E2 -10465.929} C_VEL
LIN {X 0,Y 429.311,Z 154.969,A -85,B 0,C 180,E1 -10467.44,E2 -10467.44} C_VEL
LIN {X 0,Y 424.311,Z 145.12,A -85,B 0,C 180,E1 -10468.377,E2 -10468.377} C_VEL
LIN {X 0,Y 418.912,Z 136.263,A -85,B 0,C 180,E1 -10469.424,E2 -10469.424} C_VEL
LIN {X 0,Y 416.225,Z 132.205,A -85,B 0,C 180,E1 -10469.985,E2 -10469.985} C_VEL
LIN {X 0,Y 414.228,Z 128.978,A -85,B 0,C 180,E1 -10470.455,E2 -10470.455} C_VEL
LIN {X 0,Y 412.259,Z 123.067,A -85,B 0,C 180,E1 -10473.06,E2 -10473.06} C_VEL
LIN {X 0,Y 411.206,Z 119.89,A -85,B 0,C 180,E1 -10474.877,E2 -10474.877} C_VEL
LIN {X 0,Y 411.194,Z 119.891,A -85,B 0,C 180,E1 -10478.166,E2 -10478.166} C_VEL
LIN {X 0,Y 411.159,Z 119.895,A -85,B 0,C 180,E1 -10481.807,E2 -10481.807} C_VEL
LIN {X 0,Y 411.173,Z 119.894,A -85,B 0,C 180,E1 -10485.509,E2 -10485.509} C_VEL
LIN {X 0,Y 411.146,Z 119.899,A -85,B 0,C 180,E1 -10488.774,E2 -10488.774} C_VEL
LIN {X 0,Y 411.155,Z 120.03,A -85,B 0,C 180,E1 -10489.602,E2 -10489.602} C_VEL
LIN {X 0,Y 412.615,Z 124.153,A -85,B 0,C 180,E1 -10491.583,E2 -10491.583} C_VEL
LIN {X 0,Y 414.865,Z 130.353,A -85,B 0,C 180,E1 -10493.971,E2 -10493.971} C_VEL
LIN {X 0,Y 417.139,Z 137.573,A -85,B 0,C 180,E1 -10496.221,E2 -10496.221} C_VEL
LIN {X 0,Y 419.256,Z 145.957,A -85,B 0,C 180,E1 -10498.41,E2 -10498.41} C_VEL
LIN {X 0,Y 420.518,Z 152.505,A -85,B 0,C 180,E1 -10499.909,E2 -10499.909} C_VEL
LIN {X 0,Y 420.282,Z 155.554,A -85,B 0,C 180,E1 -10500.434,E2 -10500.434} C_VEL
LIN {X 0,Y 423.58,Z 170.608,A -85,B 0,C 180,E1 -10501.391,E2 -10501.391} C_VEL
LIN {X 0,Y 426.324,Z 186.91,A -85,B 0,C 180,E1 -10502.262,E2 -10502.262} C_VEL
LIN {X 0,Y 427.663,Z 199.684,A -85,B 0,C 180,E1 -10502.818,E2 -10502.818} C_VEL
LIN {X 0,Y 423.4,Z 281.775,A -85,B 0,C 180,E1 -10504.893,E2 -10504.893} C_VEL
LIN {X 0,Y 421.421,Z 328.643,A -85,B 0,C 180,E1 -10506.047,E2 -10506.047} C_VEL
LIN {X 0,Y 420.182,Z 345.469,A -85,B 0,C 180,E1 -10506.656,E2 -10506.656} C_VEL
LIN {X 0,Y 418.513,Z 367.645,A -85,B 0,C 180,E1 -10507.76,E2 -10507.76} C_VEL
LIN {X 0,Y 417.371,Z 381.99,A -85,B 0,C 180,E1 -10508.645,E2 -10508.645} C_VEL
LIN {X 0,Y 416.342,Z 394.587,A -85,B 0,C 180,E1 -10509.625,E2 -10509.625} C_VEL
LIN {X 0,Y 415.065,Z 407.548,A -85,B 0,C 180,E1 -10510.849,E2 -10510.849} C_VEL
LIN {X 0,Y 413.95,Z 419.363,A -85,B 0,C 180,E1 -10512.206,E2 -10512.206} C_VEL
LIN {X 0,Y 412.842,Z 430.154,A -85,B 0,C 180,E1 -10513.687,E2 -10513.687} C_VEL
LIN {X 0,Y 411.877,Z 440.638,A -85,B 0,C 180,E1 -10515.423,E2 -10515.423} C_VEL
LIN {X 0,Y 411.112,Z 449.32,A -85,B 0,C 180,E1 -10517.16,E2 -10517.16} C_VEL
LIN {X 0,Y 410.73,Z 455.608,A -85,B 0,C 180,E1 -10518.651,E2 -10518.651} C_VEL
LIN {X 0,Y 410.251,Z 462.449,A -85,B 0,C 180,E1 -10520.634,E2 -10520.634} C_VEL
LIN {X 0,Y 410.112,Z 467.794,A -85,B 0,C 180,E1 -10522.616,E2 -10522.616} C_VEL
LIN {X 0,Y 409.996,Z 470.854,A -85,B 0,C 180,E1 -10524.097,E2 -10524.097} C_VEL
LIN {X 0,Y 409.931,Z 473.861,A -85,B 0,C 180,E1 -10526.068,E2 -10526.068} C_VEL
LIN {X 0,Y 410.031,Z 475.649,A -85,B 0,C 180,E1 -10528.035,E2 -10528.035} C_VEL
LIN {X 0,Y 409.93,Z 476.244,A -85,B 0,C 180,E1 -10530,E2 -10530} C_VEL
LIN {X 0,Y 410.03,Z 475.626,A -85,B 0,C 180,E1 -10531.965,E2 -10531.965} C_VEL
LIN {X 0,Y 409.937,Z 473.791,A -85,B 0,C 180,E1 -10533.932,E2 -10533.932} C_VEL
LIN {X 0,Y 410.013,Z 470.725,A -85,B 0,C 180,E1 -10535.903,E2 -10535.903} C_VEL
LIN {X 0,Y 410.132,Z 466.353,A -85,B 0,C 180,E1 -10537.879,E2 -10537.879} C_VEL
LIN {X 0,Y 410.306,Z 460.567,A -85,B 0,C 180,E1 -10539.863,E2 -10539.863} C_VEL
LIN {X 0,Y 410.757,Z 454.223,A -85,B 0,C 180,E1 -10541.598,E2 -10541.598} C_VEL
LIN {X 0,Y 411.261,Z 446.75,A -85,B 0,C 180,E1 -10543.288,E2 -10543.288} C_VEL
LIN {X 0,Y 412.054,Z 437.162,A -85,B 0,C 180,E1 -10545.076,E2 -10545.076} C_VEL
LIN {X 0,Y 412.951,Z 427.623,A -85,B 0,C 180,E1 -10546.563,E2 -10546.563} C_VEL
LIN {X 0,Y 413.948,Z 416.188,A -85,B 0,C 180,E1 -10548.054,E2 -10548.054} C_VEL
LIN {X 0,Y 414.986,Z 404.919,A -85,B 0,C 180,E1 -10549.284,E2 -10549.284} C_VEL
LIN {X 0,Y 416.106,Z 392.725,A -85,B 0,C 180,E1 -10550.387,E2 -10550.387} C_VEL
LIN {X 0,Y 417.176,Z 379.522,A -85,B 0,C 180,E1 -10551.365,E2 -10551.365} C_VEL
LIN {X 0,Y 418.22,Z 365.909,A -85,B 0,C 180,E1 -10552.163,E2 -10552.163} C_VEL
LIN {X 0,Y 418.976,Z 351.328,A -85,B 0,C 180,E1 -10552.824,E2 -10552.824} C_VEL
LIN {X 0,Y 420.213,Z 333.683,A -85,B 0,C 180,E1 -10553.535,E2 -10553.535} C_VEL
LIN {X 0,Y 421.101,Z 316.689,A -85,B 0,C 180,E1 -10554.005,E2 -10554.005} C_VEL
LIN {X 0,Y 424.275,Z 244.479,A -85,B 0,C 180,E1 -10555.77,E2 -10555.77} C_VEL
LIN {X 0,Y 426.922,Z 193.664,A -85,B 0,C 180,E1 -10557.101,E2 -10557.101} C_VEL
LIN {X 0,Y 424.748,Z 170.445,A -85,B 0,C 180,E1 -10558.115,E2 -10558.115} C_VEL
LIN {X 0,Y 422.272,Z 152.134,A -85,B 0,C 180,E1 -10559.06,E2 -10559.06} C_VEL
LIN {X 0,Y 418.745,Z 142.594,A -85,B 0,C 180,E1 -10559.935,E2 -10559.935} C_VEL
LIN {X 0,Y 412.63,Z 124.982,A -85,B 0,C 180,E1 -10561.961,E2 -10561.961} C_VEL
LIN {X 0,Y 411.222,Z 119.886,A -85,B 0,C 180,E1 -10562.662,E2 -10562.662} C_VEL
LIN {X 0,Y 411.177,Z 119.891,A -85,B 0,C 180,E1 -10565.531,E2 -10565.531} C_VEL
LIN {X 0,Y 411.178,Z 119.893,A -85,B 0,C 180,E1 -10569.229,E2 -10569.229} C_VEL
LIN {X 0,Y 411.165,Z 119.893,A -85,B 0,C 180,E1 -10572.694,E2 -10572.694} C_VEL
LIN {X 0,Y 411.163,Z 119.889,A -85,B 0,C 180,E1 -10575.882,E2 -10575.882} C_VEL
LIN {X 0,Y 411.157,Z 119.893,A -85,B 0,C 180,E1 -10579.493,E2 -10579.493} C_VEL
LIN {X 0,Y 411.185,Z 119.893,A -85,B 0,C 180,E1 -10582.026,E2 -10582.026} C_VEL
LIN {X 0,Y 411.202,Z 119.89,A -85,B 0,C 180,E1 -10585.123,E2 -10585.123} C_VEL
LIN {X 0,Y 411.184,Z 120.032,A -85,B 0,C 180,E1 -10588.256,E2 -10588.256} C_VEL
LIN {X 0,Y 412.044,Z 122.478,A -85,B 0,C 180,E1 -10588.871,E2 -10588.871} C_VEL
LIN {X 0,Y 413.47,Z 125.421,A -85,B 0,C 180,E1 -10589.552,E2 -10589.552} C_VEL
LIN {X 0,Y 417.515,Z 131.455,A -85,B 0,C 180,E1 -10590.421,E2 -10590.421} C_VEL
LIN {X 0,Y 421.958,Z 138.843,A -85,B 0,C 180,E1 -10591.31,E2 -10591.31} C_VEL
LIN {X 0,Y 427.048,Z 148.462,A -85,B 0,C 180,E1 -10592.277,E2 -10592.277} C_VEL
LIN {X 0,Y 429.202,Z 153.375,A -85,B 0,C 180,E1 -10592.691,E2 -10592.691} C_VEL
LIN {X 0,Y 424.385,Z 237.716,A -85,B 0,C 180,E1 -10594.857,E2 -10594.857} C_VEL
LIN {X 0,Y 422.175,Z 289.509,A -85,B 0,C 180,E1 -10596.146,E2 -10596.146} C_VEL
LIN {X 0,Y 421.303,Z 306.222,A -85,B 0,C 180,E1 -10596.764,E2 -10596.764} C_VEL
LIN {X 0,Y 420.355,Z 320.975,A -85,B 0,C 180,E1 -10597.515,E2 -10597.515} C_VEL
LIN {X 0,Y 419.371,Z 334.215,A -85,B 0,C 180,E1 -10598.366,E2 -10598.366} C_VEL
LIN {X 0,Y 418.157,Z 348.086,A -85,B 0,C 180,E1 -10599.461,E2 -10599.461} C_VEL
LIN {X 0,Y 416.94,Z 360.573,A -85,B 0,C 180,E1 -10600.656,E2 -10600.656} C_VEL
LIN {X 0,Y 415.838,Z 370.534,A -85,B 0,C 180,E1 -10601.78,E2 -10601.78} C_VEL
LIN {X 0,Y 414.649,Z 381.594,A -85,B 0,C 180,E1 -10603.254,E2 -10603.254} C_VEL
LIN {X 0,Y 413.586,Z 392.351,A -85,B 0,C 180,E1 -10604.981,E2 -10604.981} C_VEL
LIN {X 0,Y 412.549,Z 401.26,A -85,B 0,C 180,E1 -10606.704,E2 -10606.704} C_VEL
LIN {X 0,Y 411.897,Z 407.61,A -85,B 0,C 180,E1 -10608.185,E2 -10608.185} C_VEL
LIN {X 0,Y 411.281,Z 414.615,A -85,B 0,C 180,E1 -10610.161,E2 -10610.161} C_VEL
LIN {X 0,Y 410.766,Z 420.07,A -85,B 0,C 180,E1 -10612.133,E2 -10612.133} C_VEL
LIN {X 0,Y 410.416,Z 424.116,A -85,B 0,C 180,E1 -10614.103,E2 -10614.103} C_VEL
LIN {X 0,Y 410.326,Z 426.846,A -85,B 0,C 180,E1 -10616.072,E2 -10616.072} C_VEL
LIN {X 0,Y 410.133,Z 428.344,A -85,B 0,C 180,E1 -10618.036,E2 -10618.036} C_VEL
LIN {X 0,Y 410.029,Z 428.616,A -85,B 0,C 180,E1 -10620,E2 -10620} C_VEL
LIN {X 0,Y 410.085,Z 427.656,A -85,B 0,C 180,E1 -10621.965,E2 -10621.965} C_VEL
LIN {X 0,Y 410.194,Z 426.713,A -85,B 0,C 180,E1 -10622.947,E2 -10622.947} C_VEL
LIN {X 0,Y 410.173,Z 423.891,A -85,B 0,C 180,E1 -10624.915,E2 -10624.915} C_VEL
LIN {X 0,Y 410.394,Z 419.738,A -85,B 0,C 180,E1 -10626.885,E2 -10626.885} C_VEL
LIN {X 0,Y 410.676,Z 414.17,A -85,B 0,C 180,E1 -10628.86,E2 -10628.86} C_VEL
LIN {X 0,Y 411.062,Z 407.024,A -85,B 0,C 180,E1 -10630.84,E2 -10630.84} C_VEL
LIN {X 0,Y 411.66,Z 399.326,A -85,B 0,C 180,E1 -10632.573,E2 -10632.573} C_VEL
LIN {X 0,Y 412.201,Z 391.427,A -85,B 0,C 180,E1 -10634.062,E2 -10634.062} C_VEL
LIN {X 0,Y 412.923,Z 382.157,A -85,B 0,C 180,E1 -10635.55,E2 -10635.55} C_VEL
LIN {X 0,Y 413.816,Z 371.197,A -85,B 0,C 180,E1 -10637.036,E2 -10637.036} C_VEL
LIN {X 0,Y 414.726,Z 359.399,A -85,B 0,C 180,E1 -10638.38,E2 -10638.38} C_VEL
LIN {X 0,Y 415.76,Z 346.206,A -85,B 0,C 180,E1 -10639.632,E2 -10639.632} C_VEL
LIN {X 0,Y 416.569,Z 333.626,A -85,B 0,C 180,E1 -10640.621,E2 -10640.621} C_VEL
LIN {X 0,Y 417.522,Z 319.185,A -85,B 0,C 180,E1 -10641.541,E2 -10641.541} C_VEL
LIN {X 0,Y 418.218,Z 304.572,A -85,B 0,C 180,E1 -10642.274,E2 -10642.274} C_VEL
LIN {X 0,Y 418.81,Z 289.55,A -85,B 0,C 180,E1 -10642.834,E2 -10642.834} C_VEL
LIN {X 0,Y 419.285,Z 272.346,A -85,B 0,C 180,E1 -10643.263,E2 -10643.263} C_VEL
LIN {X 0,Y 422.577,Z 148.922,A -85,B 0,C 180,E1 -10645.846,E2 -10645.846} C_VEL
LIN {X 0,Y 422.209,Z 146.91,A -85,B 0,C 180,E1 -10645.912,E2 -10645.912} C_VEL
LIN {X 0,Y 415.172,Z 129.465,A -85,B 0,C 180,E1 -10646.71,E2 -10646.71} C_VEL
LIN {X 0,Y 411.346,Z 120.694,A -85,B 0,C 180,E1 -10647.139,E2 -10647.139} C_VEL
LIN {X 0,Y 411.177,Z 119.894,A -85,B 0,C 180,E1 -10647.206,E2 -10647.206} C_VEL
LIN {X 0,Y 411.199,Z 119.892,A -85,B 0,C 180,E1 -10649.713,E2 -10649.713} C_VEL
LIN {X 0,Y 411.206,Z 119.889,A -85,B 0,C 180,E1 -10653.156,E2 -10653.156} C_VEL
LIN {X 0,Y 411.193,Z 119.887,A -85,B 0,C 180,E1 -10656.553,E2 -10656.553} C_VEL
LIN {X 0,Y 411.171,Z 119.894,A -85,B 0,C 180,E1 -10659.721,E2 -10659.721} C_VEL
LIN {X 0,Y 411.165,Z 119.895,A -85,B 0,C 180,E1 -10663.135,E2 -10663.135} C_VEL
LIN {X 0,Y 411.166,Z 119.872,A -85,B 0,C 180,E1 -10665.882,E2 -10665.882} C_VEL
LIN {X 0,Y 411.165,Z 119.894,A -85,B 0,C 180,E1 -10669.494,E2 -10669.494} C_VEL
LIN {X 0,Y 411.19,Z 119.885,A -85,B 0,C 180,E1 -10672.026,E2 -10672.026} C_VEL
LIN {X 0,Y 411.195,Z 119.884,A -85,B 0,C 180,E1 -10675.665,E2 -10675.665} C_VEL
LIN {X 0,Y 411.189,Z 119.884,A -85,B 0,C 180,E1 -10679.152,E2 -10679.152} C_VEL
LIN {X 0,Y 411.181,Z 119.885,A -85,B 0,C 180,E1 -10681.407,E2 -10681.407} C_VEL
LIN {X 0,Y 411.215,Z 119.88,A -85,B 0,C 180,E1 -10684.934,E2 -10684.934} C_VEL
LIN {X 0,Y 411.205,Z 119.887,A -85,B 0,C 180,E1 -10687.913,E2 -10687.913} C_VEL
LIN {X 0,Y 411.218,Z 119.886,A -85,B 0,C 180,E1 -10691.051,E2 -10691.051} C_VEL
LIN {X 0,Y 411.213,Z 119.882,A -85,B 0,C 180,E1 -10694.13,E2 -10694.13} C_VEL
LIN {X 0,Y 411.307,Z 119.873,A -85,B 0,C 180,E1 -10697.166,E2 -10697.166} C_VEL
LIN {X 0,Y 411.285,Z 119.877,A -85,B 0,C 180,E1 -10700.161,E2 -10700.161} C_VEL
LIN {X 0,Y 411.391,Z 119.866,A -85,B 0,C 180,E1 -10703.132,E2 -10703.132} C_VEL
LIN {X 0,Y 411.318,Z 119.874,A -85,B 0,C 180,E1 -10704.76,E2 -10704.76} C_VEL
LIN {X 0,Y 411.079,Z 120.509,A -85,B 0,C 180,E1 -10705.293,E2 -10705.293} C_VEL
LIN {X 0,Y 410.297,Z 123.136,A -85,B 0,C 180,E1 -10706.026,E2 -10706.026} C_VEL
LIN {X 0,Y 409.36,Z 126.857,A -85,B 0,C 180,E1 -10706.68,E2 -10706.68} C_VEL
LIN {X 0,Y 408.358,Z 134.032,A -85,B 0,C 180,E1 -10707.717,E2 -10707.717} C_VEL
LIN {X 0,Y 408.769,Z 137.93,A -85,B 0,C 180,E1 -10708.362,E2 -10708.362} C_VEL
LIN {X 0,Y 409.966,Z 143.279,A -85,B 0,C 180,E1 -10709.279,E2 -10709.279} C_VEL
LIN {X 0,Y 412.869,Z 150.941,A -85,B 0,C 180,E1 -10709.63,E2 -10709.63} C_VEL
LIN {X 0,Y 417.523,Z 172.965,A -85,B 0,C 180,E1 -10710.368,E2 -10710.368} C_VEL
LIN {X 0,Y 414.825,Z 310.218,A -85,B 0,C 180,E1 -10712.822,E2 -10712.822} C_VEL
LIN {X 0,Y 414.194,Z 325.491,A -85,B 0,C 180,E1 -10713.283,E2 -10713.283} C_VEL
LIN {X 0,Y 413.404,Z 339.75,A -85,B 0,C 180,E1 -10713.899,E2 -10713.899} C_VEL
LIN {X 0,Y 412.424,Z 353.008,A -85,B 0,C 180,E1 -10714.643,E2 -10714.643} C_VEL
LIN {X 0,Y 411.314,Z 366.931,A -85,B 0,C 180,E1 -10715.638,E2 -10715.638} C_VEL
LIN {X 0,Y 410.125,Z 379.148,A -85,B 0,C 180,E1 -10716.705,E2 -10716.705} C_VEL
LIN {X 0,Y 408.807,Z 391.679,A -85,B 0,C 180,E1 -10718.029,E2 -10718.029} C_VEL
LIN {X 0,Y 407.59,Z 402.698,A -85,B 0,C 180,E1 -10719.428,E2 -10719.428} C_VEL
LIN {X 0,Y 406.479,Z 412.844,A -85,B 0,C 180,E1 -10720.964,E2 -10720.964} C_VEL
LIN {X 0,Y 405.402,Z 422.801,A -85,B 0,C 180,E1 -10722.77,E2 -10722.77} C_VEL
LIN {X 0,Y 404.541,Z 431.067,A -85,B 0,C 180,E1 -10724.59,E2 -10724.59} C_VEL
LIN {X 0,Y 403.885,Z 438.109,A -85,B 0,C 180,E1 -10726.488,E2 -10726.488} C_VEL
LIN {X 0,Y 403.454,Z 443.444,A -85,B 0,C 180,E1 -10728.273,E2 -10728.273} C_VEL
LIN {X 0,Y 403.099,Z 448.422,A -85,B 0,C 180,E1 -10730.408,E2 -10730.408} C_VEL
LIN {X 0,Y 402.803,Z 451.999,A -85,B 0,C 180,E1 -10732.572,E2 -10732.572} C_VEL
LIN {X 0,Y 402.66,Z 454.237,A -85,B 0,C 180,E1 -10734.823,E2 -10734.823} C_VEL
LIN {X 0,Y 402.641,Z 455.019,A -85,B 0,C 180,E1 -10737.102,E2 -10737.102} C_VEL
LIN {X 0,Y 402.674,Z 454.387,A -85,B 0,C 180,E1 -10739.255,E2 -10739.255} C_VEL
LIN {X 0,Y 402.806,Z 452.601,A -85,B 0,C 180,E1 -10741.247,E2 -10741.247} C_VEL
LIN {X 0,Y 403.037,Z 449.769,A -85,B 0,C 180,E1 -10743.174,E2 -10743.174} C_VEL
LIN {X 0,Y 403.341,Z 445.809,A -85,B 0,C 180,E1 -10745.1,E2 -10745.1} C_VEL
LIN {X 0,Y 403.787,Z 440.355,A -85,B 0,C 180,E1 -10747.115,E2 -10747.115} C_VEL
LIN {X 0,Y 404.425,Z 433.73,A -85,B 0,C 180,E1 -10749.046,E2 -10749.046} C_VEL
LIN {X 0,Y 405.248,Z 425.747,A -85,B 0,C 180,E1 -10750.936,E2 -10750.936} C_VEL
LIN {X 0,Y 406.355,Z 416.391,A -85,B 0,C 180,E1 -10752.753,E2 -10752.753} C_VEL
LIN {X 0,Y 407.622,Z 405.741,A -85,B 0,C 180,E1 -10754.462,E2 -10754.462} C_VEL
LIN {X 0,Y 408.943,Z 393.924,A -85,B 0,C 180,E1 -10756.034,E2 -10756.034} C_VEL
LIN {X 0,Y 410.252,Z 382.378,A -85,B 0,C 180,E1 -10757.305,E2 -10757.305} C_VEL
LIN {X 0,Y 411.644,Z 368.959,A -85,B 0,C 180,E1 -10758.526,E2 -10758.526} C_VEL
LIN {X 0,Y 412.874,Z 355.412,A -85,B 0,C 180,E1 -10759.524,E2 -10759.524} C_VEL
LIN {X 0,Y 413.913,Z 342.215,A -85,B 0,C 180,E1 -10760.298,E2 -10760.298} C_VEL
LIN {X 0,Y 414.802,Z 326.922,A -85,B 0,C 180,E1 -10760.986,E2 -10760.986} C_VEL
LIN {X 0,Y 415.522,Z 311.328,A -85,B 0,C 180,E1 -10761.467,E2 -10761.467} C_VEL
LIN {X 0,Y 416.766,Z 251.18,A -85,B 0,C 180,E1 -10762.57,E2 -10762.57} C_VEL
LIN {X 0,Y 418.484,Z 167.697,A -85,B 0,C 180,E1 -10764.074,E2 -10764.074} C_VEL
LIN {X 0,Y 415.969,Z 154.061,A -85,B 0,C 180,E1 -10764.531,E2 -10764.531} C_VEL
LIN {X 0,Y 410.794,Z 142.119,A -85,B 0,C 180,E1 -10765.18,E2 -10765.18} C_VEL
LIN {X 0,Y 407.559,Z 131.068,A -85,B 0,C 180,E1 -10766.804,E2 -10766.804} C_VEL
LIN {X 0,Y 404.151,Z 120.765,A -85,B 0,C 180,E1 -10768.407,E2 -10768.407} C_VEL
LIN {X 0,Y 404.198,Z 120.763,A -85,B 0,C 180,E1 -10772,E2 -10772} C_VEL
LIN {X 0,Y 404.229,Z 120.759,A -85,B 0,C 180,E1 -10772.461,E2 -10772.461} C_VEL
LIN {X 0,Y 405.247,Z 123.624,A -85,B 0,C 180,E1 -10772.617,E2 -10772.617} C_VEL
LIN {X 0,Y 414.891,Z 146.244,A -85,B 0,C 180,E1 -10773.72,E2 -10773.72} C_VEL
LIN {X 0,Y 416.15,Z 149.678,A -85,B 0,C 180,E1 -10773.871,E2 -10773.871} C_VEL
LIN {X 0,Y 412.251,Z 285.388,A -85,B 0,C 180,E1 -10776.815,E2 -10776.815} C_VEL
LIN {X 0,Y 411.681,Z 300.872,A -85,B 0,C 180,E1 -10777.347,E2 -10777.347} C_VEL
LIN {X 0,Y 410.903,Z 316.542,A -85,B 0,C 180,E1 -10778.094,E2 -10778.094} C_VEL
LIN {X 0,Y 410.075,Z 329.843,A -85,B 0,C 180,E1 -10778.905,E2 -10778.905} C_VEL
LIN {X 0,Y 409.132,Z 343.17,A -85,B 0,C 180,E1 -10779.906,E2 -10779.906} C_VEL
LIN {X 0,Y 408.147,Z 356.621,A -85,B 0,C 180,E1 -10781.141,E2 -10781.141} C_VEL
LIN {X 0,Y 407.108,Z 369.272,A -85,B 0,C 180,E1 -10782.545,E2 -10782.545} C_VEL
LIN {X 0,Y 406.259,Z 379.794,A -85,B 0,C 180,E1 -10783.931,E2 -10783.931} C_VEL
LIN {X 0,Y 405.423,Z 389.501,A -85,B 0,C 180,E1 -10785.442,E2 -10785.442} C_VEL
LIN {X 0,Y 404.704,Z 399.014,A -85,B 0,C 180,E1 -10787.208,E2 -10787.208} C_VEL
LIN {X 0,Y 404.075,Z 406.878,A -85,B 0,C 180,E1 -10788.97,E2 -10788.97} C_VEL
LIN {X 0,Y 403.638,Z 414.203,A -85,B 0,C 180,E1 -10790.984,E2 -10790.984} C_VEL
LIN {X 0,Y 403.307,Z 419.924,A -85,B 0,C 180,E1 -10792.993,E2 -10792.993} C_VEL
LIN {X 0,Y 403.126,Z 424.199,A -85,B 0,C 180,E1 -10794.999,E2 -10794.999} C_VEL
LIN {X 0,Y 403.142,Z 427.147,A -85,B 0,C 180,E1 -10797.002,E2 -10797.002} C_VEL
LIN {X 0,Y 402.958,Z 428.855,A -85,B 0,C 180,E1 -10799,E2 -10799} C_VEL
LIN {X 0,Y 402.997,Z 429.33,A -85,B 0,C 180,E1 -10800.999,E2 -10800.999} C_VEL
LIN {X 0,Y 403.181,Z 428.574,A -85,B 0,C 180,E1 -10802.997,E2 -10802.997} C_VEL
LIN {X 0,Y 403.286,Z 427.739,A -85,B 0,C 180,E1 -10803.997,E2 -10803.997} C_VEL
LIN {X 0,Y 403.392,Z 425.145,A -85,B 0,C 180,E1 -10806,E2 -10806} C_VEL
LIN {X 0,Y 403.764,Z 421.231,A -85,B 0,C 180,E1 -10808.004,E2 -10808.004} C_VEL
LIN {X 0,Y 404.368,Z 415.925,A -85,B 0,C 180,E1 -10810.009,E2 -10810.009} C_VEL
LIN {X 0,Y 405.023,Z 409.09,A -85,B 0,C 180,E1 -10812.018,E2 -10812.018} C_VEL
LIN {X 0,Y 405.812,Z 401.756,A -85,B 0,C 180,E1 -10813.765,E2 -10813.765} C_VEL
LIN {X 0,Y 406.958,Z 392.753,A -85,B 0,C 180,E1 -10815.526,E2 -10815.526} C_VEL
LIN {X 0,Y 408.174,Z 381.981,A -85,B 0,C 180,E1 -10817.278,E2 -10817.278} C_VEL
LIN {X 0,Y 409.454,Z 370.89,A -85,B 0,C 180,E1 -10818.773,E2 -10818.773} C_VEL
LIN {X 0,Y 410.799,Z 358.758,A -85,B 0,C 180,E1 -10820.139,E2 -10820.139} C_VEL
LIN {X 0,Y 412.142,Z 345.531,A -85,B 0,C 180,E1 -10821.376,E2 -10821.376} C_VEL
LIN {X 0,Y 413.455,Z 330.93,A -85,B 0,C 180,E1 -10822.486,E2 -10822.486} C_VEL
LIN {X 0,Y 414.625,Z 316.35,A -85,B 0,C 180,E1 -10823.369,E2 -10823.369} C_VEL
LIN {X 0,Y 415.735,Z 300.045,A -85,B 0,C 180,E1 -10824.119,E2 -10824.119} C_VEL
LIN {X 0,Y 416.447,Z 284.969,A -85,B 0,C 180,E1 -10824.625,E2 -10824.625} C_VEL
LIN {X 0,Y 419.988,Z 216.544,A -85,B 0,C 180,E1 -10826.391,E2 -10826.391} C_VEL
LIN {X 0,Y 423.767,Z 157.671,A -85,B 0,C 180,E1 -10827.988,E2 -10827.988} C_VEL
LIN {X 0,Y 419.125,Z 148.566,A -85,B 0,C 180,E1 -10828.911,E2 -10828.911} C_VEL
LIN {X 0,Y 414.373,Z 140.663,A -85,B 0,C 180,E1 -10829.901,E2 -10829.901} C_VEL
LIN {X 0,Y 409.822,Z 133.86,A -85,B 0,C 180,E1 -10830.912,E2 -10830.912} C_VEL
LIN {X 0,Y 407.337,Z 130.185,A -85,B 0,C 180,E1 -10831.541,E2 -10831.541} C_VEL
LIN {X 0,Y 405.825,Z 125.651,A -85,B 0,C 180,E1 -10833.772,E2 -10833.772} C_VEL
LIN {X 0,Y 404.875,Z 123.133,A -85,B 0,C 180,E1 -10835.329,E2 -10835.329} C_VEL
LIN {X 0,Y 404.139,Z 120.77,A -85,B 0,C 180,E1 -10837.141,E2 -10837.141} C_VEL
LIN {X 0,Y 404.116,Z 120.773,A -85,B 0,C 180,E1 -10840.075,E2 -10840.075} C_VEL
LIN {X 0,Y 404.141,Z 120.77,A -85,B 0,C 180,E1 -10843.082,E2 -10843.082} C_VEL
LIN {X 0,Y 404.119,Z 120.771,A -85,B 0,C 180,E1 -10845.922,E2 -10845.922} C_VEL
LIN {X 0,Y 404.147,Z 120.807,A -85,B 0,C 180,E1 -10847.297,E2 -10847.297} C_VEL
LIN {X 0,Y 405.681,Z 125.309,A -85,B 0,C 180,E1 -10850.135,E2 -10850.135} C_VEL
LIN {X 0,Y 407.586,Z 130.375,A -85,B 0,C 180,E1 -10852.483,E2 -10852.483} C_VEL
LIN {X 0,Y 409.215,Z 135.214,A -85,B 0,C 180,E1 -10854.273,E2 -10854.273} C_VEL
LIN {X 0,Y 411.119,Z 141.48,A -85,B 0,C 180,E1 -10856.25,E2 -10856.25} C_VEL
LIN {X 0,Y 413.276,Z 150.598,A -85,B 0,C 180,E1 -10858.642,E2 -10858.642} C_VEL
LIN {X 0,Y 414.039,Z 154.569,A -85,B 0,C 180,E1 -10859.543,E2 -10859.543} C_VEL
LIN {X 0,Y 416.149,Z 162.359,A -85,B 0,C 180,E1 -10860.155,E2 -10860.155} C_VEL
LIN {X 0,Y 419.182,Z 178.228,A -85,B 0,C 180,E1 -10861.144,E2 -10861.144} C_VEL
LIN {X 0,Y 421.278,Z 192.638,A -85,B 0,C 180,E1 -10861.899,E2 -10861.899} C_VEL
LIN {X 0,Y 422.019,Z 200.289,A -85,B 0,C 180,E1 -10862.243,E2 -10862.243} C_VEL
LIN {X 0,Y 417.346,Z 282.855,A -85,B 0,C 180,E1 -10864.403,E2 -10864.403} C_VEL
LIN {X 0,Y 415.328,Z 327.503,A -85,B 0,C 180,E1 -10865.54,E2 -10865.54} C_VEL
LIN {X 0,Y 413.993,Z 344.381,A -85,B 0,C 180,E1 -10866.156,E2 -10866.156} C_VEL
LIN {X 0,Y 412.62,Z 359.976,A -85,B 0,C 180,E1 -10866.936,E2 -10866.936} C_VEL
LIN {X 0,Y 411.092,Z 378.543,A -85,B 0,C 180,E1 -10868.039,E2 -10868.039} C_VEL
LIN {X 0,Y 409.899,Z 391.75,A -85,B 0,C 180,E1 -10869.028,E2 -10869.028} C_VEL
LIN {X 0,Y 408.57,Z 405.162,A -85,B 0,C 180,E1 -10870.271,E2 -10870.271} C_VEL
LIN {X 0,Y 407.425,Z 416.754,A -85,B 0,C 180,E1 -10871.575,E2 -10871.575} C_VEL
LIN {X 0,Y 406.156,Z 428.408,A -85,B 0,C 180,E1 -10873.152,E2 -10873.152} C_VEL
LIN {X 0,Y 405.218,Z 437.766,A -85,B 0,C 180,E1 -10874.663,E2 -10874.663} C_VEL
LIN {X 0,Y 404.342,Z 447.152,A -85,B 0,C 180,E1 -10876.48,E2 -10876.48} C_VEL
LIN {X 0,Y 403.705,Z 455.463,A -85,B 0,C 180,E1 -10878.451,E2 -10878.451} C_VEL
LIN {X 0,Y 403.187,Z 462.296,A -85,B 0,C 180,E1 -10880.468,E2 -10880.468} C_VEL
LIN {X 0,Y 403.027,Z 467.634,A -85,B 0,C 180,E1 -10882.485,E2 -10882.485} C_VEL
LIN {X 0,Y 402.936,Z 470.69,A -85,B 0,C 180,E1 -10883.993,E2 -10883.993} C_VEL
LIN {X 0,Y 402.849,Z 473.688,A -85,B 0,C 180,E1 -10885.998,E2 -10885.998} C_VEL
LIN {X 0,Y 402.939,Z 475.469,A -85,B 0,C 180,E1 -10888.001,E2 -10888.001} C_VEL
LIN {X 0,Y 402.854,Z 476.057,A -85,B 0,C 180,E1 -10890,E2 -10890} C_VEL
LIN {X 0,Y 402.938,Z 475.435,A -85,B 0,C 180,E1 -10891.999,E2 -10891.999} C_VEL
LIN {X 0,Y 402.854,Z 473.591,A -85,B 0,C 180,E1 -10894.001,E2 -10894.001} C_VEL
LIN {X 0,Y 402.976,Z 470.111,A -85,B 0,C 180,E1 -10896.232,E2 -10896.232} C_VEL
LIN {X 0,Y 403.042,Z 466.131,A -85,B 0,C 180,E1 -10898.019,E2 -10898.019} C_VEL
LIN {X 0,Y 403.249,Z 460.33,A -85,B 0,C 180,E1 -10900.037,E2 -10900.037} C_VEL
LIN {X 0,Y 403.712,Z 453.969,A -85,B 0,C 180,E1 -10901.803,E2 -10901.803} C_VEL
LIN {X 0,Y 404.281,Z 446.232,A -85,B 0,C 180,E1 -10903.573,E2 -10903.573} C_VEL
LIN {X 0,Y 405.126,Z 436.875,A -85,B 0,C 180,E1 -10905.34,E2 -10905.34} C_VEL
LIN {X 0,Y 406.079,Z 427.316,A -85,B 0,C 180,E1 -10906.851,E2 -10906.851} C_VEL
LIN {X 0,Y 407.04,Z 416.755,A -85,B 0,C 180,E1 -10908.262,E2 -10908.262} C_VEL
LIN {X 0,Y 408.215,Z 404.562,A -85,B 0,C 180,E1 -10909.616,E2 -10909.616} C_VEL
LIN {X 0,Y 409.416,Z 392.348,A -85,B 0,C 180,E1 -10910.735,E2 -10910.735} C_VEL
LIN {X 0,Y 410.523,Z 379.101,A -85,B 0,C 180,E1 -10911.729,E2 -10911.729} C_VEL
LIN {X 0,Y 411.671,Z 364.782,A -85,B 0,C 180,E1 -10912.573,E2 -10912.573} C_VEL
LIN {X 0,Y 413.277,Z 343.321,A -85,B 0,C 180,E1 -10913.622,E2 -10913.622} C_VEL
LIN {X 0,Y 414.382,Z 327.771,A -85,B 0,C 180,E1 -10914.186,E2 -10914.186} C_VEL
LIN {X 0,Y 419.056,Z 233.161,A -85,B 0,C 180,E1 -10916.622,E2 -10916.622} C_VEL
LIN {X 0,Y 421.275,Z 194.993,A -85,B 0,C 180,E1 -10917.656,E2 -10917.656} C_VEL
LIN {X 0,Y 419.346,Z 172.546,A -85,B 0,C 180,E1 -10918.671,E2 -10918.671} C_VEL
LIN {X 0,Y 417.181,Z 155.358,A -85,B 0,C 180,E1 -10919.593,E2 -10919.593} C_VEL
LIN {X 0,Y 412.975,Z 144.093,A -85,B 0,C 180,E1 -10920.665,E2 -10920.665} C_VEL
LIN {X 0,Y 407.697,Z 127.697,A -85,B 0,C 180,E1 -10922.644,E2 -10922.644} C_VEL
LIN {X 0,Y 407.275,Z 126.251,A -85,B 0,C 180,E1 -10922.831,E2 -10922.831} C_VEL
LIN {X 0,Y 404.86,Z 123.111,A -85,B 0,C 180,E1 -10923.568,E2 -10923.568} C_VEL
LIN {X 0,Y 404.139,Z 120.768,A -85,B 0,C 180,E1 -10923.963,E2 -10923.963} C_VEL
LIN {X 0,Y 404.136,Z 120.77,A -85,B 0,C 180,E1 -10927.492,E2 -10927.492} C_VEL
LIN {X 0,Y 404.115,Z 120.771,A -85,B 0,C 180,E1 -10930.075,E2 -10930.075} C_VEL
LIN {X 0,Y 404.14,Z 120.769,A -85,B 0,C 180,E1 -10933.082,E2 -10933.082} C_VEL
LIN {X 0,Y 404.12,Z 120.766,A -85,B 0,C 180,E1 -10935.922,E2 -10935.922} C_VEL
LIN {X 0,Y 404.101,Z 120.773,A -85,B 0,C 180,E1 -10938.633,E2 -10938.633} C_VEL
LIN {X 0,Y 404.139,Z 120.77,A -85,B 0,C 180,E1 -10941.495,E2 -10941.495} C_VEL
LIN {X 0,Y 404.173,Z 120.767,A -85,B 0,C 180,E1 -10944.983,E2 -10944.983} C_VEL
LIN {X 0,Y 404.156,Z 120.774,A -85,B 0,C 180,E1 -10946.981,E2 -10946.981} C_VEL
LIN {X 0,Y 405.017,Z 123.424,A -85,B 0,C 180,E1 -10947.662,E2 -10947.662} C_VEL
LIN {X 0,Y 406.171,Z 125.462,A -85,B 0,C 180,E1 -10948.252,E2 -10948.252} C_VEL
LIN {X 0,Y 406.997,Z 127.055,A -85,B 0,C 180,E1 -10948.555,E2 -10948.555} C_VEL
LIN {X 0,Y 411.664,Z 133.638,A -85,B 0,C 180,E1 -10949.635,E2 -10949.635} C_VEL
LIN {X 0,Y 417.052,Z 142.562,A -85,B 0,C 180,E1 -10950.799,E2 -10950.799} C_VEL
LIN {X 0,Y 422.765,Z 153.697,A -85,B 0,C 180,E1 -10951.955,E2 -10951.955} C_VEL
LIN {X 0,Y 423.6,Z 156.253,A -85,B 0,C 180,E1 -10952.148,E2 -10952.148} C_VEL
LIN {X 0,Y 418.526,Z 237.767,A -85,B 0,C 180,E1 -10954.314,E2 -10954.314} C_VEL
LIN {X 0,Y 416.048,Z 290.302,A -85,B 0,C 180,E1 -10955.666,E2 -10955.666} C_VEL
LIN {X 0,Y 415.172,Z 306.137,A -85,B 0,C 180,E1 -10956.266,E2 -10956.266} C_VEL
LIN {X 0,Y 414.138,Z 320.981,A -85,B 0,C 180,E1 -10957.026,E2 -10957.026} C_VEL
LIN {X 0,Y 413.075,Z 334.204,A -85,B 0,C 180,E1 -10957.887,E2 -10957.887} C_VEL
LIN {X 0,Y 411.75,Z 348.147,A -85,B 0,C 180,E1 -10958.996,E2 -10958.996} C_VEL
LIN {X 0,Y 410.366,Z 361.676,A -85,B 0,C 180,E1 -10960.321,E2 -10960.321} C_VEL
LIN {X 0,Y 409.189,Z 371.656,A -85,B 0,C 180,E1 -10961.474,E2 -10961.474} C_VEL
LIN {X 0,Y 407.916,Z 382.597,A -85,B 0,C 180,E1 -10962.969,E2 -10962.969} C_VEL
LIN {X 0,Y 406.785,Z 393.225,A -85,B 0,C 180,E1 -10964.724,E2 -10964.724} C_VEL
LIN {X 0,Y 405.672,Z 402.124,A -85,B 0,C 180,E1 -10966.49,E2 -10966.49} C_VEL
LIN {X 0,Y 404.836,Z 410.248,A -85,B 0,C 180,E1 -10968.484,E2 -10968.484} C_VEL
LIN {X 0,Y 404.183,Z 416.781,A -85,B 0,C 180,E1 -10970.492,E2 -10970.492} C_VEL
LIN {X 0,Y 403.675,Z 421.816,A -85,B 0,C 180,E1 -10972.497,E2 -10972.497} C_VEL
LIN {X 0,Y 403.376,Z 424.685,A -85,B 0,C 180,E1 -10974,E2 -10974} C_VEL
LIN {X 0,Y 403.269,Z 427.357,A -85,B 0,C 180,E1 -10976.003,E2 -10976.003} C_VEL
LIN {X 0,Y 403.061,Z 428.799,A -85,B 0,C 180,E1 -10978.002,E2 -10978.002} C_VEL
LIN {X 0,Y 402.949,Z 429.01,A -85,B 0,C 180,E1 -10980,E2 -10980} C_VEL
LIN {X 0,Y 403.016,Z 427.983,A -85,B 0,C 180,E1 -10981.999,E2 -10981.999} C_VEL
LIN {X 0,Y 403.066,Z 425.721,A -85,B 0,C 180,E1 -10984,E2 -10984} C_VEL
LIN {X 0,Y 403.249,Z 422.166,A -85,B 0,C 180,E1 -10986.003,E2 -10986.003} C_VEL
LIN {X 0,Y 403.442,Z 417.238,A -85,B 0,C 180,E1 -10988.011,E2 -10988.011} C_VEL
LIN {X 0,Y 403.796,Z 410.804,A -85,B 0,C 180,E1 -10990.024,E2 -10990.024} C_VEL
LIN {X 0,Y 404.431,Z 402.671,A -85,B 0,C 180,E1 -10992.037,E2 -10992.037} C_VEL
LIN {X 0,Y 404.99,Z 393.986,A -85,B 0,C 180,E1 -10993.799,E2 -10993.799} C_VEL
LIN {X 0,Y 405.852,Z 383.426,A -85,B 0,C 180,E1 -10995.57,E2 -10995.57} C_VEL
LIN {X 0,Y 406.764,Z 372.621,A -85,B 0,C 180,E1 -10997.081,E2 -10997.081} C_VEL
LIN {X 0,Y 407.65,Z 361.537,A -85,B 0,C 180,E1 -10998.393,E2 -10998.393} C_VEL
LIN {X 0,Y 408.769,Z 348.064,A -85,B 0,C 180,E1 -10999.72,E2 -10999.72} C_VEL
LIN {X 0,Y 409.698,Z 334.091,A -85,B 0,C 180,E1 -11000.852,E2 -11000.852} C_VEL
LIN {X 0,Y 410.671,Z 319.687,A -85,B 0,C 180,E1 -11001.787,E2 -11001.787} C_VEL
LIN {X 0,Y 411.45,Z 304.255,A -85,B 0,C 180,E1 -11002.571,E2 -11002.571} C_VEL
LIN {X 0,Y 412.078,Z 288.357,A -85,B 0,C 180,E1 -11003.162,E2 -11003.162} C_VEL
LIN {X 0,Y 412.598,Z 270.421,A -85,B 0,C 180,E1 -11003.597,E2 -11003.597} C_VEL
LIN {X 0,Y 415.958,Z 149.894,A -85,B 0,C 180,E1 -11006.185,E2 -11006.185} C_VEL
LIN {X 0,Y 409.546,Z 133.498,A -85,B 0,C 180,E1 -11006.935,E2 -11006.935} C_VEL
LIN {X 0,Y 404.232,Z 121.243,A -85,B 0,C 180,E1 -11007.54,E2 -11007.54} C_VEL
LIN {X 0,Y 404.136,Z 120.769,A -85,B 0,C 180,E1 -11007.589,E2 -11007.589} C_VEL
LIN {X 0,Y 404.146,Z 120.769,A -85,B 0,C 180,E1 -11010.286,E2 -11010.286} C_VEL
LIN {X 0,Y 404.14,Z 120.77,A -85,B 0,C 180,E1 -11013.813,E2 -11013.813} C_VEL
LIN {X 0,Y 404.136,Z 120.767,A -85,B 0,C 180,E1 -11016.875,E2 -11016.875} C_VEL
LIN {X 0,Y 404.119,Z 120.77,A -85,B 0,C 180,E1 -11020.075,E2 -11020.075} C_VEL
LIN {X 0,Y 404.145,Z 120.769,A -85,B 0,C 180,E1 -11023.082,E2 -11023.082} C_VEL
LIN {X 0,Y 404.122,Z 120.749,A -85,B 0,C 180,E1 -11025.922,E2 -11025.922} C_VEL
LIN {X 0,Y 404.105,Z 120.763,A -85,B 0,C 180,E1 -11028.633,E2 -11028.633} C_VEL
LIN {X 0,Y 404.144,Z 120.766,A -85,B 0,C 180,E1 -11031.495,E2 -11031.495} C_VEL
LIN {X 0,Y 404.176,Z 120.748,A -85,B 0,C 180,E1 -11034.983,E2 -11034.983} C_VEL
LIN {X 0,Y 404.14,Z 120.768,A -85,B 0,C 180,E1 -11038.443,E2 -11038.443} C_VEL
LIN {X 0,Y 404.154,Z 120.755,A -85,B 0,C 180,E1 -11040.863,E2 -11040.863} C_VEL
LIN {X 0,Y 404.143,Z 120.768,A -85,B 0,C 180,E1 -11044.231,E2 -11044.231} C_VEL
LIN {X 0,Y 404.168,Z 120.763,A -85,B 0,C 180,E1 -11047.508,E2 -11047.508} C_VEL
LIN {X 0,Y 404.163,Z 120.761,A -85,B 0,C 180,E1 -11050.707,E2 -11050.707} C_VEL
LIN {X 0,Y 404.183,Z 120.757,A -85,B 0,C 180,E1 -11053.847,E2 -11053.847} C_VEL
LIN {X 0,Y 404.287,Z 120.747,A -85,B 0,C 180,E1 -11056.939,E2 -11056.939} C_VEL
LIN {X 0,Y 404.252,Z 120.751,A -85,B 0,C 180,E1 -11059.988,E2 -11059.988} C_VEL
LIN {X 0,Y 404.342,Z 120.745,A -85,B 0,C 180,E1 -11063.012,E2 -11063.012} C_VEL
LIN {X 0,Y 404.248,Z 120.918,A -85,B 0,C 180,E1 -11065.357,E2 -11065.357} C_VEL
LIN {X 0,Y 407.491,Z 132.288,A -85,B 0,C 180,E1 -11067.381,E2 -11067.381} C_VEL
LIN {X 0,Y 408.769,Z 137.93,A -85,B 0,C 180,E1 -11068.362,E2 -11068.362} C_VEL
LIN {X 0,Y 409.237,Z 140.724,A -85,B 0,C 180,E1 -11068.733,E2 -11068.733} C_VEL
LIN {X 0,Y 409.467,Z 145.876,A -85,B 0,C 180,E1 -11069.127,E2 -11069.127} C_VEL
LIN {X 0,Y 409.381,Z 151.574,A -85,B 0,C 180,E1 -11069.369,E2 -11069.369} C_VEL
LIN {X 0,Y 409.478,Z 163.907,A -85,B 0,C 180,E1 -11069.652,E2 -11069.652} C_VEL
LIN {X 0,Y 409.882,Z 167.969,A -85,B 0,C 180,E1 -11069.76,E2 -11069.76} C_VEL
LIN {X 0,Y 411.116,Z 174.203,A -85,B 0,C 180,E1 -11069.966,E2 -11069.966} C_VEL
LIN {X 0,Y 408.33,Z 309.468,A -85,B 0,C 180,E1 -11072.414,E2 -11072.414} C_VEL
LIN {X 0,Y 407.653,Z 325.076,A -85,B 0,C 180,E1 -11072.881,E2 -11072.881} C_VEL
LIN {X 0,Y 406.838,Z 339.863,A -85,B 0,C 180,E1 -11073.528,E2 -11073.528} C_VEL
LIN {X 0,Y 405.717,Z 354.1,A -85,B 0,C 180,E1 -11074.346,E2 -11074.346} C_VEL
LIN {X 0,Y 404.556,Z 367.871,A -85,B 0,C 180,E1 -11075.358,E2 -11075.358} C_VEL
LIN {X 0,Y 403.221,Z 380.926,A -85,B 0,C 180,E1 -11076.537,E2 -11076.537} C_VEL
LIN {X 0,Y 401.838,Z 393.461,A -85,B 0,C 180,E1 -11077.917,E2 -11077.917} C_VEL
LIN {X 0,Y 400.596,Z 404.256,A -85,B 0,C 180,E1 -11079.339,E2 -11079.339} C_VEL
LIN {X 0,Y 399.463,Z 414.079,A -85,B 0,C 180,E1 -11080.876,E2 -11080.876} C_VEL
LIN {X 0,Y 398.498,Z 422.683,A -85,B 0,C 180,E1 -11082.477,E2 -11082.477} C_VEL
LIN {X 0,Y 397.567,Z 431.006,A -85,B 0,C 180,E1 -11084.329,E2 -11084.329} C_VEL
LIN {X 0,Y 396.993,Z 436.946,A -85,B 0,C 180,E1 -11085.926,E2 -11085.926} C_VEL
LIN {X 0,Y 396.411,Z 443.467,A -85,B 0,C 180,E1 -11088.075,E2 -11088.075} C_VEL
LIN {X 0,Y 396.081,Z 447.73,A -85,B 0,C 180,E1 -11089.876,E2 -11089.876} C_VEL
LIN {X 0,Y 395.8,Z 451.326,A -85,B 0,C 180,E1 -11091.894,E2 -11091.894} C_VEL
LIN {X 0,Y 395.583,Z 453.898,A -85,B 0,C 180,E1 -11094.118,E2 -11094.118} C_VEL
LIN {X 0,Y 395.559,Z 454.665,A -85,B 0,C 180,E1 -11095.24,E2 -11095.24} C_VEL
LIN {X 0,Y 395.54,Z 455.156,A -85,B 0,C 180,E1 -11097.514,E2 -11097.514} C_VEL
LIN {X 0,Y 395.588,Z 454.194,A -85,B 0,C 180,E1 -11099.831,E2 -11099.831} C_VEL
LIN {X 0,Y 395.758,Z 452.584,A -85,B 0,C 180,E1 -11101.525,E2 -11101.525} C_VEL
LIN {X 0,Y 396.083,Z 448.705,A -85,B 0,C 180,E1 -11103.987,E2 -11103.987} C_VEL
LIN {X 0,Y 396.419,Z 444.709,A -85,B 0,C 180,E1 -11105.806,E2 -11105.806} C_VEL
LIN {X 0,Y 396.964,Z 438.499,A -85,B 0,C 180,E1 -11107.973,E2 -11107.973} C_VEL
LIN {X 0,Y 397.795,Z 430.863,A -85,B 0,C 180,E1 -11110.061,E2 -11110.061} C_VEL
LIN {X 0,Y 398.82,Z 421.91,A -85,B 0,C 180,E1 -11112.039,E2 -11112.039} C_VEL
LIN {X 0,Y 399.929,Z 413.285,A -85,B 0,C 180,E1 -11113.623,E2 -11113.623} C_VEL
LIN {X 0,Y 401.157,Z 403.114,A -85,B 0,C 180,E1 -11115.197,E2 -11115.197} C_VEL
LIN {X 0,Y 402.664,Z 390.757,A -85,B 0,C 180,E1 -11116.777,E2 -11116.777} C_VEL
LIN {X 0,Y 404.012,Z 379.191,A -85,B 0,C 180,E1 -11118.007,E2 -11118.007} C_VEL
LIN {X 0,Y 405.307,Z 366.622,A -85,B 0,C 180,E1 -11119.118,E2 -11119.118} C_VEL
LIN {X 0,Y 406.651,Z 352.081,A -85,B 0,C 180,E1 -11120.15,E2 -11120.15} C_VEL
LIN {X 0,Y 407.776,Z 337.59,A -85,B 0,C 180,E1 -11120.95,E2 -11120.95} C_VEL
LIN {X 0,Y 408.636,Z 322.451,A -85,B 0,C 180,E1 -11121.572,E2 -11121.572} C_VEL
LIN {X 0,Y 409.235,Z 308.174,A -85,B 0,C 180,E1 -11121.971,E2 -11121.971} C_VEL
LIN {X 0,Y 412.304,Z 169.284,A -85,B 0,C 180,E1 -11124.505,E2 -11124.505} C_VEL
LIN {X 0,Y 410.059,Z 156.813,A -85,B 0,C 180,E1 -11124.93,E2 -11124.93} C_VEL
LIN {X 0,Y 403.708,Z 142.202,A -85,B 0,C 180,E1 -11125.77,E2 -11125.77} C_VEL
LIN {X 0,Y 399.648,Z 129.14,A -85,B 0,C 180,E1 -11127.751,E2 -11127.751} C_VEL
LIN {X 0,Y 397.098,Z 121.646,A -85,B 0,C 180,E1 -11128.934,E2 -11128.934} C_VEL
LIN {X 0,Y 397.156,Z 121.64,A -85,B 0,C 180,E1 -11132.082,E2 -11132.082} C_VEL
LIN {X 0,Y 399.017,Z 126.532,A -85,B 0,C 180,E1 -11132.318,E2 -11132.318} C_VEL
LIN {X 0,Y 408.492,Z 148.507,A -85,B 0,C 180,E1 -11133.415,E2 -11133.415} C_VEL
LIN {X 0,Y 409.465,Z 150.982,A -85,B 0,C 180,E1 -11133.529,E2 -11133.529} C_VEL
LIN {X 0,Y 405.455,Z 286.002,A -85,B 0,C 180,E1 -11136.539,E2 -11136.539} C_VEL
LIN {X 0,Y 404.844,Z 301.873,A -85,B 0,C 180,E1 -11137.103,E2 -11137.103} C_VEL
LIN {X 0,Y 404.067,Z 316.937,A -85,B 0,C 180,E1 -11137.838,E2 -11137.838} C_VEL
LIN {X 0,Y 403.202,Z 330.216,A -85,B 0,C 180,E1 -11138.662,E2 -11138.662} C_VEL
LIN {X 0,Y 402.237,Z 343.541,A -85,B 0,C 180,E1 -11139.68,E2 -11139.68} C_VEL
LIN {X 0,Y 401.159,Z 357.583,A -85,B 0,C 180,E1 -11140.997,E2 -11140.997} C_VEL
LIN {X 0,Y 400.157,Z 369.664,A -85,B 0,C 180,E1 -11142.364,E2 -11142.364} C_VEL
LIN {X 0,Y 399.19,Z 381.043,A -85,B 0,C 180,E1 -11143.901,E2 -11143.901} C_VEL
LIN {X 0,Y 398.351,Z 390.668,A -85,B 0,C 180,E1 -11145.439,E2 -11145.439} C_VEL
LIN {X 0,Y 397.659,Z 400.059,A -85,B 0,C 180,E1 -11147.237,E2 -11147.237} C_VEL
LIN {X 0,Y 396.982,Z 407.847,A -85,B 0,C 180,E1 -11149.029,E2 -11149.029} C_VEL
LIN {X 0,Y 396.587,Z 414.227,A -85,B 0,C 180,E1 -11150.822,E2 -11150.822} C_VEL
LIN {X 0,Y 396.237,Z 420.049,A -85,B 0,C 180,E1 -11152.868,E2 -11152.868} C_VEL
LIN {X 0,Y 396.065,Z 424.416,A -85,B 0,C 180,E1 -11154.91,E2 -11154.91} C_VEL
LIN {X 0,Y 396.058,Z 427.448,A -85,B 0,C 180,E1 -11156.948,E2 -11156.948} C_VEL
LIN {X 0,Y 395.883,Z 429.228,A -85,B 0,C 180,E1 -11158.982,E2 -11158.982} C_VEL
LIN {X 0,Y 395.921,Z 429.772,A -85,B 0,C 180,E1 -11161.017,E2 -11161.017} C_VEL
LIN {X 0,Y 396.122,Z 429.082,A -85,B 0,C 180,E1 -11163.051,E2 -11163.051} C_VEL
LIN {X 0,Y 396.232,Z 428.277,A -85,B 0,C 180,E1 -11164.068,E2 -11164.068} C_VEL
LIN {X 0,Y 396.359,Z 425.746,A -85,B 0,C 180,E1 -11166.107,E2 -11166.107} C_VEL
LIN {X 0,Y 396.773,Z 421.887,A -85,B 0,C 180,E1 -11168.146,E2 -11168.146} C_VEL
LIN {X 0,Y 397.405,Z 416.64,A -85,B 0,C 180,E1 -11170.186,E2 -11170.186} C_VEL
LIN {X 0,Y 398.115,Z 409.893,A -85,B 0,C 180,E1 -11172.23,E2 -11172.23} C_VEL
LIN {X 0,Y 398.961,Z 402.648,A -85,B 0,C 180,E1 -11173.998,E2 -11173.998} C_VEL
LIN {X 0,Y 400.173,Z 393.7,A -85,B 0,C 180,E1 -11175.796,E2 -11175.796} C_VEL
LIN {X 0,Y 401.498,Z 383.07,A -85,B 0,C 180,E1 -11177.575,E2 -11177.575} C_VEL
LIN {X 0,Y 402.954,Z 371.105,A -85,B 0,C 180,E1 -11179.22,E2 -11179.22} C_VEL
LIN {X 0,Y 404.386,Z 358.961,A -85,B 0,C 180,E1 -11180.605,E2 -11180.605} C_VEL
LIN {X 0,Y 405.861,Z 345.726,A -85,B 0,C 180,E1 -11181.857,E2 -11181.857} C_VEL
LIN {X 0,Y 407.272,Z 331.153,A -85,B 0,C 180,E1 -11182.981,E2 -11182.981} C_VEL
LIN {X 0,Y 408.53,Z 316.365,A -85,B 0,C 180,E1 -11183.888,E2 -11183.888} C_VEL
LIN {X 0,Y 409.685,Z 300.73,A -85,B 0,C 180,E1 -11184.622,E2 -11184.622} C_VEL
LIN {X 0,Y 410.443,Z 285.74,A -85,B 0,C 180,E1 -11185.142,E2 -11185.142} C_VEL
LIN {X 0,Y 414.509,Z 214.588,A -85,B 0,C 180,E1 -11187.039,E2 -11187.039} C_VEL
LIN {X 0,Y 418.329,Z 160.354,A -85,B 0,C 180,E1 -11188.564,E2 -11188.564} C_VEL
LIN {X 0,Y 413.472,Z 150.952,A -85,B 0,C 180,E1 -11189.6,E2 -11189.6} C_VEL
LIN {X 0,Y 408.615,Z 143.074,A -85,B 0,C 180,E1 -11190.686,E2 -11190.686} C_VEL
LIN {X 0,Y 405.671,Z 138.778,A -85,B 0,C 180,E1 -11191.391,E2 -11191.391} C_VEL
LIN {X 0,Y 402.943,Z 135.005,A -85,B 0,C 180,E1 -11192.078,E2 -11192.078} C_VEL
LIN {X 0,Y 400.547,Z 131.462,A -85,B 0,C 180,E1 -11192.785,E2 -11192.785} C_VEL
LIN {X 0,Y 399.658,Z 128.778,A -85,B 0,C 180,E1 -11194.259,E2 -11194.259} C_VEL
LIN {X 0,Y 398.376,Z 125.147,A -85,B 0,C 180,E1 -11196.856,E2 -11196.856} C_VEL
LIN {X 0,Y 397.372,Z 122.988,A -85,B 0,C 180,E1 -11199.546,E2 -11199.546} C_VEL
LIN {X 0,Y 397.163,Z 122.182,A -85,B 0,C 180,E1 -11201.994,E2 -11201.994} C_VEL
LIN {X 0,Y 397.237,Z 122.461,A -85,B 0,C 180,E1 -11203.63,E2 -11203.63} C_VEL
LIN {X 0,Y 397.973,Z 124.292,A -85,B 0,C 180,E1 -11206.471,E2 -11206.471} C_VEL
LIN {X 0,Y 398.645,Z 125.993,A -85,B 0,C 180,E1 -11207.938,E2 -11207.938} C_VEL
LIN {X 0,Y 399.764,Z 128.991,A -85,B 0,C 180,E1 -11209.883,E2 -11209.883} C_VEL
LIN {X 0,Y 401.559,Z 133.816,A -85,B 0,C 180,E1 -11212.225,E2 -11212.225} C_VEL
LIN {X 0,Y 403.284,Z 139.234,A -85,B 0,C 180,E1 -11214.291,E2 -11214.291} C_VEL
LIN {X 0,Y 405.195,Z 145.739,A -85,B 0,C 180,E1 -11216.361,E2 -11216.361} C_VEL
LIN {X 0,Y 407.009,Z 153.601,A -85,B 0,C 180,E1 -11218.433,E2 -11218.433} C_VEL
LIN {X 0,Y 409.865,Z 159.91,A -85,B 0,C 180,E1 -11219.161,E2 -11219.161} C_VEL
LIN {X 0,Y 412.052,Z 169.712,A -85,B 0,C 180,E1 -11219.884,E2 -11219.884} C_VEL
LIN {X 0,Y 414.838,Z 186.342,A -85,B 0,C 180,E1 -11220.906,E2 -11220.906} C_VEL
LIN {X 0,Y 416.428,Z 201.086,A -85,B 0,C 180,E1 -11221.639,E2 -11221.639} C_VEL
LIN {X 0,Y 411.662,Z 278.747,A -85,B 0,C 180,E1 -11223.751,E2 -11223.751} C_VEL
LIN {X 0,Y 409.236,Z 326.831,A -85,B 0,C 180,E1 -11225.016,E2 -11225.016} C_VEL
LIN {X 0,Y 407.882,Z 343.529,A -85,B 0,C 180,E1 -11225.641,E2 -11225.641} C_VEL
LIN {X 0,Y 406.488,Z 358.121,A -85,B 0,C 180,E1 -11226.374,E2 -11226.374} C_VEL
LIN {X 0,Y 404.18,Z 382.108,A -85,B 0,C 180,E1 -11227.912,E2 -11227.912} C_VEL
LIN {X 0,Y 403.002,Z 394.606,A -85,B 0,C 180,E1 -11228.919,E2 -11228.919} C_VEL
LIN {X 0,Y 401.576,Z 407.478,A -85,B 0,C 180,E1 -11230.179,E2 -11230.179} C_VEL
LIN {X 0,Y 400.331,Z 419.224,A -85,B 0,C 180,E1 -11231.579,E2 -11231.579} C_VEL
LIN {X 0,Y 399.126,Z 429.963,A -85,B 0,C 180,E1 -11233.11,E2 -11233.11} C_VEL
LIN {X 0,Y 398.016,Z 440.404,A -85,B 0,C 180,E1 -11234.903,E2 -11234.903} C_VEL
LIN {X 0,Y 397.117,Z 449.256,A -85,B 0,C 180,E1 -11236.746,E2 -11236.746} C_VEL
LIN {X 0,Y 396.534,Z 457.146,A -85,B 0,C 180,E1 -11238.758,E2 -11238.758} C_VEL
LIN {X 0,Y 396.063,Z 463.585,A -85,B 0,C 180,E1 -11240.81,E2 -11240.81} C_VEL
LIN {X 0,Y 395.909,Z 468.553,A -85,B 0,C 180,E1 -11242.862,E2 -11242.862} C_VEL
LIN {X 0,Y 395.795,Z 472.177,A -85,B 0,C 180,E1 -11244.906,E2 -11244.906} C_VEL
LIN {X 0,Y 395.747,Z 474.551,A -85,B 0,C 180,E1 -11246.946,E2 -11246.946} C_VEL
LIN {X 0,Y 395.8,Z 475.727,A -85,B 0,C 180,E1 -11248.983,E2 -11248.983} C_VEL
LIN {X 0,Y 395.799,Z 475.711,A -85,B 0,C 180,E1 -11251.017,E2 -11251.017} C_VEL
LIN {X 0,Y 395.747,Z 474.465,A -85,B 0,C 180,E1 -11253.054,E2 -11253.054} C_VEL
LIN {X 0,Y 395.799,Z 472.004,A -85,B 0,C 180,E1 -11255.094,E2 -11255.094} C_VEL
LIN {X 0,Y 395.908,Z 468.273,A -85,B 0,C 180,E1 -11257.138,E2 -11257.138} C_VEL
LIN {X 0,Y 396.043,Z 463.184,A -85,B 0,C 180,E1 -11259.19,E2 -11259.19} C_VEL
LIN {X 0,Y 396.498,Z 456.608,A -85,B 0,C 180,E1 -11261.243,E2 -11261.243} C_VEL
LIN {X 0,Y 397.048,Z 448.333,A -85,B 0,C 180,E1 -11263.303,E2 -11263.303} C_VEL
LIN {X 0,Y 397.912,Z 439.453,A -85,B 0,C 180,E1 -11265.101,E2 -11265.101} C_VEL
LIN {X 0,Y 398.87,Z 430.365,A -85,B 0,C 180,E1 -11266.638,E2 -11266.638} C_VEL
LIN {X 0,Y 399.913,Z 419.031,A -85,B 0,C 180,E1 -11268.251,E2 -11268.251} C_VEL
LIN {X 0,Y 401.074,Z 407.775,A -85,B 0,C 180,E1 -11269.58,E2 -11269.58} C_VEL
LIN {X 0,Y 402.421,Z 394.823,A -85,B 0,C 180,E1 -11270.845,E2 -11270.845} C_VEL
LIN {X 0,Y 403.568,Z 382.204,A -85,B 0,C 180,E1 -11271.854,E2 -11271.854} C_VEL
LIN {X 0,Y 404.801,Z 367.834,A -85,B 0,C 180,E1 -11272.765,E2 -11272.765} C_VEL
LIN {X 0,Y 406.291,Z 351.528,A -85,B 0,C 180,E1 -11273.714,E2 -11273.714} C_VEL
LIN {X 0,Y 407.719,Z 335.104,A -85,B 0,C 180,E1 -11274.437,E2 -11274.437} C_VEL
LIN {X 0,Y 408.766,Z 318.882,A -85,B 0,C 180,E1 -11274.947,E2 -11274.947} C_VEL
LIN {X 0,Y 412.877,Z 241.301,A -85,B 0,C 180,E1 -11276.984,E2 -11276.984} C_VEL
LIN {X 0,Y 415.717,Z 195.957,A -85,B 0,C 180,E1 -11278.253,E2 -11278.253} C_VEL
LIN {X 0,Y 414.004,Z 173.958,A -85,B 0,C 180,E1 -11279.294,E2 -11279.294} C_VEL
LIN {X 0,Y 412.244,Z 158.709,A -85,B 0,C 180,E1 -11280.138,E2 -11280.138} C_VEL
LIN {X 0,Y 407.94,Z 146.981,A -85,B 0,C 180,E1 -11281.293,E2 -11281.293} C_VEL
LIN {X 0,Y 404.852,Z 137.427,A -85,B 0,C 180,E1 -11282.438,E2 -11282.438} C_VEL
LIN {X 0,Y 403.157,Z 131.519,A -85,B 0,C 180,E1 -11283.201,E2 -11283.201} C_VEL
LIN {X 0,Y 401.115,Z 128.776,A -85,B 0,C 180,E1 -11283.851,E2 -11283.851} C_VEL
LIN {X 0,Y 399.952,Z 126.475,A -85,B 0,C 180,E1 -11284.322,E2 -11284.322} C_VEL
LIN {X 0,Y 398.371,Z 124.87,A -85,B 0,C 180,E1 -11284.843,E2 -11284.843} C_VEL
LIN {X 0,Y 397.647,Z 123.622,A -85,B 0,C 180,E1 -11285.154,E2 -11285.154} C_VEL
LIN {X 0,Y 397.093,Z 121.645,A -85,B 0,C 180,E1 -11285.528,E2 -11285.528} C_VEL
LIN {X 0,Y 397.092,Z 121.645,A -85,B 0,C 180,E1 -11288.855,E2 -11288.855} C_VEL
LIN {X 0,Y 397.053,Z 121.648,A -85,B 0,C 180,E1 -11292.269,E2 -11292.269} C_VEL
LIN {X 0,Y 397.084,Z 121.645,A -85,B 0,C 180,E1 -11295.069,E2 -11295.069} C_VEL
LIN {X 0,Y 397.05,Z 121.65,A -85,B 0,C 180,E1 -11298.024,E2 -11298.024} C_VEL
LIN {X 0,Y 397.091,Z 121.649,A -85,B 0,C 180,E1 -11301.724,E2 -11301.724} C_VEL
LIN {X 0,Y 397.111,Z 121.72,A -85,B 0,C 180,E1 -11305.474,E2 -11305.474} C_VEL
LIN {X 0,Y 397.828,Z 124.029,A -85,B 0,C 180,E1 -11306.13,E2 -11306.13} C_VEL
LIN {X 0,Y 399.436,Z 126.899,A -85,B 0,C 180,E1 -11307.093,E2 -11307.093} C_VEL
LIN {X 0,Y 403.372,Z 132.497,A -85,B 0,C 180,E1 -11308.17,E2 -11308.17} C_VEL
LIN {X 0,Y 408.116,Z 139.441,A -85,B 0,C 180,E1 -11309.334,E2 -11309.334} C_VEL
LIN {X 0,Y 413.199,Z 148.27,A -85,B 0,C 180,E1 -11310.49,E2 -11310.49} C_VEL
LIN {X 0,Y 417.985,Z 157.844,A -85,B 0,C 180,E1 -11311.513,E2 -11311.513} C_VEL
LIN {X 0,Y 418.139,Z 158.875,A -85,B 0,C 180,E1 -11311.572,E2 -11311.572} C_VEL
LIN {X 0,Y 412.602,Z 240.679,A -85,B 0,C 180,E1 -11313.815,E2 -11313.815} C_VEL
LIN {X 0,Y 409.973,Z 291.95,A -85,B 0,C 180,E1 -11315.187,E2 -11315.187} C_VEL
LIN {X 0,Y 408.967,Z 308.062,A -85,B 0,C 180,E1 -11315.832,E2 -11315.832} C_VEL
LIN {X 0,Y 407.788,Z 323.22,A -85,B 0,C 180,E1 -11316.647,E2 -11316.647} C_VEL
LIN {X 0,Y 406.557,Z 337.679,A -85,B 0,C 180,E1 -11317.648,E2 -11317.648} C_VEL
LIN {X 0,Y 405.153,Z 351.011,A -85,B 0,C 180,E1 -11318.771,E2 -11318.771} C_VEL
LIN {X 0,Y 403.76,Z 363.474,A -85,B 0,C 180,E1 -11320.043,E2 -11320.043} C_VEL
LIN {X 0,Y 402.571,Z 372.862,A -85,B 0,C 180,E1 -11321.158,E2 -11321.158} C_VEL
LIN {X 0,Y 401.209,Z 383.669,A -85,B 0,C 180,E1 -11322.675,E2 -11322.675} C_VEL
LIN {X 0,Y 399.995,Z 394.152,A -85,B 0,C 180,E1 -11324.458,E2 -11324.458} C_VEL
LIN {X 0,Y 398.807,Z 403.011,A -85,B 0,C 180,E1 -11326.266,E2 -11326.266} C_VEL
LIN {X 0,Y 398.058,Z 409.151,A -85,B 0,C 180,E1 -11327.768,E2 -11327.768} C_VEL
LIN {X 0,Y 397.481,Z 414.438,A -85,B 0,C 180,E1 -11329.301,E2 -11329.301} C_VEL
LIN {X 0,Y 396.895,Z 420.129,A -85,B 0,C 180,E1 -11331.344,E2 -11331.344} C_VEL
LIN {X 0,Y 396.515,Z 423.755,A -85,B 0,C 180,E1 -11333.011,E2 -11333.011} C_VEL
LIN {X 0,Y 396.131,Z 426.744,A -85,B 0,C 180,E1 -11334.911,E2 -11334.911} C_VEL
LIN {X 0,Y 396.214,Z 427.88,A -85,B 0,C 180,E1 -11335.932,E2 -11335.932} C_VEL
LIN {X 0,Y 395.992,Z 429.26,A -85,B 0,C 180,E1 -11337.966,E2 -11337.966} C_VEL
LIN {X 0,Y 395.871,Z 429.403,A -85,B 0,C 180,E1 -11340,E2 -11340} C_VEL
LIN {X 0,Y 395.949,Z 428.305,A -85,B 0,C 180,E1 -11342.035,E2 -11342.035} C_VEL
LIN {X 0,Y 395.977,Z 425.968,A -85,B 0,C 180,E1 -11344.071,E2 -11344.071} C_VEL
LIN {X 0,Y 396.171,Z 422.326,A -85,B 0,C 180,E1 -11346.11,E2 -11346.11} C_VEL
LIN {X 0,Y 396.394,Z 417.302,A -85,B 0,C 180,E1 -11348.155,E2 -11348.155} C_VEL
LIN {X 0,Y 396.771,Z 410.763,A -85,B 0,C 180,E1 -11350.203,E2 -11350.203} C_VEL
LIN {X 0,Y 397.332,Z 403.664,A -85,B 0,C 180,E1 -11351.996,E2 -11351.996} C_VEL
LIN {X 0,Y 397.908,Z 394.784,A -85,B 0,C 180,E1 -11353.845,E2 -11353.845} C_VEL
LIN {X 0,Y 398.793,Z 384.643,A -85,B 0,C 180,E1 -11355.59,E2 -11355.59} C_VEL
LIN {X 0,Y 399.697,Z 373.978,A -85,B 0,C 180,E1 -11357.129,E2 -11357.129} C_VEL
LIN {X 0,Y 400.724,Z 361.812,A -85,B 0,C 180,E1 -11358.598,E2 -11358.598} C_VEL
LIN {X 0,Y 401.876,Z 348.404,A -85,B 0,C 180,E1 -11359.939,E2 -11359.939} C_VEL
LIN {X 0,Y 402.83,Z 334.419,A -85,B 0,C 180,E1 -11361.09,E2 -11361.09} C_VEL
LIN {X 0,Y 403.84,Z 320.022,A -85,B 0,C 180,E1 -11362.04,E2 -11362.04} C_VEL
LIN {X 0,Y 404.604,Z 304.875,A -85,B 0,C 180,E1 -11362.826,E2 -11362.826} C_VEL
LIN {X 0,Y 405.27,Z 289.164,A -85,B 0,C 180,E1 -11363.427,E2 -11363.427} C_VEL
LIN {X 0,Y 405.807,Z 271.131,A -85,B 0,C 180,E1 -11363.88,E2 -11363.88} C_VEL
LIN {X 0,Y 409.328,Z 151.484,A -85,B 0,C 180,E1 -11366.514,E2 -11366.514} C_VEL
LIN {X 0,Y 403.139,Z 135.929,A -85,B 0,C 180,E1 -11367.241,E2 -11367.241} C_VEL
LIN {X 0,Y 397.206,Z 122.257,A -85,B 0,C 180,E1 -11367.942,E2 -11367.942} C_VEL
LIN {X 0,Y 397.084,Z 121.648,A -85,B 0,C 180,E1 -11367.979,E2 -11367.979} C_VEL
LIN {X 0,Y 397.079,Z 121.648,A -85,B 0,C 180,E1 -11370.883,E2 -11370.883} C_VEL
LIN {X 0,Y 397.121,Z 121.641,A -85,B 0,C 180,E1 -11374.494,E2 -11374.494} C_VEL
LIN {X 0,Y 397.094,Z 121.644,A -85,B 0,C 180,E1 -11378.277,E2 -11378.277} C_VEL
LIN {X 0,Y 397.054,Z 121.65,A -85,B 0,C 180,E1 -11381.977,E2 -11381.977} C_VEL
LIN {X 0,Y 397.087,Z 121.634,A -85,B 0,C 180,E1 -11385.069,E2 -11385.069} C_VEL
LIN {X 0,Y 397.054,Z 121.64,A -85,B 0,C 180,E1 -11388.024,E2 -11388.024} C_VEL
LIN {X 0,Y 397.096,Z 121.642,A -85,B 0,C 180,E1 -11391.724,E2 -11391.724} C_VEL
LIN {X 0,Y 397.12,Z 121.634,A -85,B 0,C 180,E1 -11395.506,E2 -11395.506} C_VEL
LIN {X 0,Y 397.078,Z 121.642,A -85,B 0,C 180,E1 -11399.117,E2 -11399.117} C_VEL
LIN {X 0,Y 397.094,Z 121.644,A -85,B 0,C 180,E1 -11402.602,E2 -11402.602} C_VEL
LIN {X 0,Y 397.114,Z 121.631,A -85,B 0,C 180,E1 -11405.98,E2 -11405.98} C_VEL
LIN {X 0,Y 397.142,Z 121.633,A -85,B 0,C 180,E1 -11409.705,E2 -11409.705} C_VEL
LIN {X 0,Y 397.157,Z 121.636,A -85,B 0,C 180,E1 -11412.859,E2 -11412.859} C_VEL
LIN {X 0,Y 397.233,Z 121.626,A -85,B 0,C 180,E1 -11416.703,E2 -11416.703} C_VEL
LIN {X 0,Y 397.214,Z 121.627,A -85,B 0,C 180,E1 -11419.809,E2 -11419.809} C_VEL
LIN {X 0,Y 397.295,Z 121.623,A -85,B 0,C 180,E1 -11422.887,E2 -11422.887} C_VEL
LIN {X 0,Y 397.261,Z 121.809,A -85,B 0,C 180,E1 -11424.925,E2 -11424.925} C_VEL
LIN {X 0,Y 401.023,Z 135.34,A -85,B 0,C 180,E1 -11427.365,E2 -11427.365} C_VEL
LIN {X 0,Y 402.905,Z 143.495,A -85,B 0,C 180,E1 -11428.781,E2 -11428.781} C_VEL
LIN {X 0,Y 406.824,Z 153.652,A -85,B 0,C 180,E1 -11429.264,E2 -11429.264} C_VEL
LIN {X 0,Y 409.882,Z 167.969,A -85,B 0,C 180,E1 -11429.76,E2 -11429.76} C_VEL
LIN {X 0,Y 410.09,Z 171.83,A -85,B 0,C 180,E1 -11429.85,E2 -11429.85} C_VEL
LIN {X 0,Y 409.66,Z 175.727,A -85,B 0,C 180,E1 -11429.898,E2 -11429.898} C_VEL
LIN {X 0,Y 407.669,Z 183.444,A -85,B 0,C 180,E1 -11429.914,E2 -11429.914} C_VEL
LIN {X 0,Y 404.874,Z 193.168,A -85,B 0,C 180,E1 -11429.915,E2 -11429.915} C_VEL
LIN {X 0,Y 404.16,Z 199.123,A -85,B 0,C 180,E1 -11429.983,E2 -11429.983} C_VEL
LIN {X 0,Y 401.788,Z 310.696,A -85,B 0,C 180,E1 -11432.046,E2 -11432.046} C_VEL
LIN {X 0,Y 401.086,Z 325.86,A -85,B 0,C 180,E1 -11432.515,E2 -11432.515} C_VEL
LIN {X 0,Y 400.268,Z 340.001,A -85,B 0,C 180,E1 -11433.145,E2 -11433.145} C_VEL
LIN {X 0,Y 399.225,Z 353.282,A -85,B 0,C 180,E1 -11433.912,E2 -11433.912} C_VEL
LIN {X 0,Y 397.984,Z 367.27,A -85,B 0,C 180,E1 -11434.939,E2 -11434.939} C_VEL
LIN {X 0,Y 396.616,Z 380.152,A -85,B 0,C 180,E1 -11436.103,E2 -11436.103} C_VEL
LIN {X 0,Y 395.276,Z 392.053,A -85,B 0,C 180,E1 -11437.406,E2 -11437.406} C_VEL
LIN {X 0,Y 393.829,Z 403.995,A -85,B 0,C 180,E1 -11438.983,E2 -11438.983} C_VEL
LIN {X 0,Y 392.611,Z 414.041,A -85,B 0,C 180,E1 -11440.573,E2 -11440.573} C_VEL
LIN {X 0,Y 391.435,Z 423.842,A -85,B 0,C 180,E1 -11442.442,E2 -11442.442} C_VEL
LIN {X 0,Y 390.58,Z 431.16,A -85,B 0,C 180,E1 -11444.113,E2 -11444.113} C_VEL
LIN {X 0,Y 389.803,Z 438.754,A -85,B 0,C 180,E1 -11446.228,E2 -11446.228} C_VEL
LIN {X 0,Y 389.245,Z 444.914,A -85,B 0,C 180,E1 -11448.419,E2 -11448.419} C_VEL
LIN {X 0,Y 388.95,Z 448.547,A -85,B 0,C 180,E1 -11450.079,E2 -11450.079} C_VEL
LIN {X 0,Y 388.64,Z 452.199,A -85,B 0,C 180,E1 -11452.319,E2 -11452.319} C_VEL
LIN {X 0,Y 388.483,Z 454.467,A -85,B 0,C 180,E1 -11454.588,E2 -11454.588} C_VEL
LIN {X 0,Y 388.426,Z 455.357,A -85,B 0,C 180,E1 -11456.894,E2 -11456.894} C_VEL
LIN {X 0,Y 388.494,Z 454.818,A -85,B 0,C 180,E1 -11459.238,E2 -11459.238} C_VEL
LIN {X 0,Y 388.668,Z 452.768,A -85,B 0,C 180,E1 -11461.627,E2 -11461.627} C_VEL
LIN {X 0,Y 388.951,Z 449.565,A -85,B 0,C 180,E1 -11463.779,E2 -11463.779} C_VEL
LIN {X 0,Y 389.388,Z 444.693,A -85,B 0,C 180,E1 -11466.067,E2 -11466.067} C_VEL
LIN {X 0,Y 389.957,Z 438.92,A -85,B 0,C 180,E1 -11468.117,E2 -11468.117} C_VEL
LIN {X 0,Y 390.74,Z 432.106,A -85,B 0,C 180,E1 -11470.05,E2 -11470.05} C_VEL
LIN {X 0,Y 391.711,Z 423.987,A -85,B 0,C 180,E1 -11471.938,E2 -11471.938} C_VEL
LIN {X 0,Y 393.064,Z 413.941,A -85,B 0,C 180,E1 -11473.856,E2 -11473.856} C_VEL
LIN {X 0,Y 394.494,Z 402.745,A -85,B 0,C 180,E1 -11475.61,E2 -11475.61} C_VEL
LIN {X 0,Y 395.906,Z 391.603,A -85,B 0,C 180,E1 -11477.064,E2 -11477.064} C_VEL
LIN {X 0,Y 397.365,Z 379.762,A -85,B 0,C 180,E1 -11478.353,E2 -11478.353} C_VEL
LIN {X 0,Y 398.827,Z 366.321,A -85,B 0,C 180,E1 -11479.556,E2 -11479.556} C_VEL
LIN {X 0,Y 400.123,Z 353.13,A -85,B 0,C 180,E1 -11480.511,E2 -11480.511} C_VEL
LIN {X 0,Y 401.324,Z 338.203,A -85,B 0,C 180,E1 -11481.356,E2 -11481.356} C_VEL
LIN {X 0,Y 402.233,Z 323.034,A -85,B 0,C 180,E1 -11481.993,E2 -11481.993} C_VEL
LIN {X 0,Y 402.915,Z 307.303,A -85,B 0,C 180,E1 -11482.432,E2 -11482.432} C_VEL
LIN {X 0,Y 406.026,Z 169.974,A -85,B 0,C 180,E1 -11484.98,E2 -11484.98} C_VEL
LIN {X 0,Y 404.1,Z 159.402,A -85,B 0,C 180,E1 -11485.354,E2 -11485.354} C_VEL
LIN {X 0,Y 396.574,Z 142.339,A -85,B 0,C 180,E1 -11486.371,E2 -11486.371} C_VEL
LIN {X 0,Y 391.822,Z 127.729,A -85,B 0,C 180,E1 -11488.656,E2 -11488.656} C_VEL
LIN {X 0,Y 390.042,Z 122.528,A -85,B 0,C 180,E1 -11489.513,E2 -11489.513} C_VEL
LIN {X 0,Y 390.109,Z 122.636,A -85,B 0,C 180,E1 -11491.674,E2 -11491.674} C_VEL
LIN {X 0,Y 392.223,Z 127.891,A -85,B 0,C 180,E1 -11491.943,E2 -11491.943} C_VEL
LIN {X 0,Y 402.257,Z 151.222,A -85,B 0,C 180,E1 -11493.126,E2 -11493.126} C_VEL
LIN {X 0,Y 402.835,Z 153.547,A -85,B 0,C 180,E1 -11493.217,E2 -11493.217} C_VEL
LIN {X 0,Y 398.699,Z 285.91,A -85,B 0,C 180,E1 -11496.236,E2 -11496.236} C_VEL
LIN {X 0,Y 398.032,Z 301.925,A -85,B 0,C 180,E1 -11496.811,E2 -11496.811} C_VEL
LIN {X 0,Y 397.238,Z 317.267,A -85,B 0,C 180,E1 -11497.574,E2 -11497.574} C_VEL
LIN {X 0,Y 396.227,Z 332.311,A -85,B 0,C 180,E1 -11498.541,E2 -11498.541} C_VEL
LIN {X 0,Y 395.135,Z 346.773,A -85,B 0,C 180,E1 -11499.706,E2 -11499.706} C_VEL
LIN {X 0,Y 394.062,Z 359.478,A -85,B 0,C 180,E1 -11500.952,E2 -11500.952} C_VEL
LIN {X 0,Y 393.022,Z 372.041,A -85,B 0,C 180,E1 -11502.436,E2 -11502.436} C_VEL
LIN {X 0,Y 391.963,Z 383.961,A -85,B 0,C 180,E1 -11504.131,E2 -11504.131} C_VEL
LIN {X 0,Y 391.072,Z 394.115,A -85,B 0,C 180,E1 -11505.868,E2 -11505.868} C_VEL
LIN {X 0,Y 390.519,Z 402.229,A -85,B 0,C 180,E1 -11507.528,E2 -11507.528} C_VEL
LIN {X 0,Y 389.883,Z 408.756,A -85,B 0,C 180,E1 -11509.089,E2 -11509.089} C_VEL
LIN {X 0,Y 389.445,Z 415.868,A -85,B 0,C 180,E1 -11511.176,E2 -11511.176} C_VEL
LIN {X 0,Y 389.184,Z 420.156,A -85,B 0,C 180,E1 -11512.738,E2 -11512.738} C_VEL
LIN {X 0,Y 389.005,Z 424.617,A -85,B 0,C 180,E1 -11514.817,E2 -11514.817} C_VEL
LIN {X 0,Y 388.977,Z 427.735,A -85,B 0,C 180,E1 -11516.892,E2 -11516.892} C_VEL
LIN {X 0,Y 388.811,Z 429.597,A -85,B 0,C 180,E1 -11518.964,E2 -11518.964} C_VEL
LIN {X 0,Y 388.847,Z 430.217,A -85,B 0,C 180,E1 -11521.035,E2 -11521.035} C_VEL
LIN {X 0,Y 389.065,Z 429.599,A -85,B 0,C 180,E1 -11523.106,E2 -11523.106} C_VEL
LIN {X 0,Y 389.178,Z 428.83,A -85,B 0,C 180,E1 -11524.142,E2 -11524.142} C_VEL
LIN {X 0,Y 389.327,Z 426.354,A -85,B 0,C 180,E1 -11526.218,E2 -11526.218} C_VEL
LIN {X 0,Y 389.76,Z 422.556,A -85,B 0,C 180,E1 -11528.294,E2 -11528.294} C_VEL
LIN {X 0,Y 390.431,Z 417.378,A -85,B 0,C 180,E1 -11530.37,E2 -11530.37} C_VEL
LIN {X 0,Y 391.231,Z 410.718,A -85,B 0,C 180,E1 -11532.448,E2 -11532.448} C_VEL
LIN {X 0,Y 392.134,Z 403.476,A -85,B 0,C 180,E1 -11534.266,E2 -11534.266} C_VEL
LIN {X 0,Y 393.411,Z 394.719,A -85,B 0,C 180,E1 -11536.075,E2 -11536.075} C_VEL
LIN {X 0,Y 394.573,Z 385.826,A -85,B 0,C 180,E1 -11537.625,E2 -11537.625} C_VEL
LIN {X 0,Y 396.015,Z 375.312,A -85,B 0,C 180,E1 -11539.166,E2 -11539.166} C_VEL
LIN {X 0,Y 397.434,Z 364.587,A -85,B 0,C 180,E1 -11540.498,E2 -11540.498} C_VEL
LIN {X 0,Y 398.958,Z 351.667,A -85,B 0,C 180,E1 -11541.847,E2 -11541.847} C_VEL
LIN {X 0,Y 400.502,Z 338.382,A -85,B 0,C 180,E1 -11542.982,E2 -11542.982} C_VEL
LIN {X 0,Y 401.822,Z 324.72,A -85,B 0,C 180,E1 -11543.945,E2 -11543.945} C_VEL
LIN {X 0,Y 403.039,Z 310.511,A -85,B 0,C 180,E1 -11544.74,E2 -11544.74} C_VEL
LIN {X 0,Y 404.153,Z 294.465,A -85,B 0,C 180,E1 -11545.423,E2 -11545.423} C_VEL
LIN {X 0,Y 405.354,Z 271.474,A -85,B 0,C 180,E1 -11546.1,E2 -11546.1} C_VEL
LIN {X 0,Y 409.991,Z 201.572,A -85,B 0,C 180,E1 -11548.048,E2 -11548.048} C_VEL
LIN {X 0,Y 412.992,Z 163.113,A -85,B 0,C 180,E1 -11549.166,E2 -11549.166} C_VEL
LIN {X 0,Y 408.428,Z 154.41,A -85,B 0,C 180,E1 -11550.203,E2 -11550.203} C_VEL
LIN {X 0,Y 404.125,Z 147.373,A -85,B 0,C 180,E1 -11551.242,E2 -11551.242} C_VEL
LIN {X 0,Y 399.769,Z 141.016,A -85,B 0,C 180,E1 -11552.374,E2 -11552.374} C_VEL
LIN {X 0,Y 396.733,Z 136.883,A -85,B 0,C 180,E1 -11553.246,E2 -11553.246} C_VEL
LIN {X 0,Y 393.833,Z 132.925,A -85,B 0,C 180,E1 -11554.203,E2 -11554.203} C_VEL
LIN {X 0,Y 392.732,Z 129.905,A -85,B 0,C 180,E1 -11556.362,E2 -11556.362} C_VEL
LIN {X 0,Y 392.116,Z 128.265,A -85,B 0,C 180,E1 -11557.943,E2 -11557.943} C_VEL
LIN {X 0,Y 391.532,Z 126.872,A -85,B 0,C 180,E1 -11560.255,E2 -11560.255} C_VEL
LIN {X 0,Y 391.475,Z 126.51,A -85,B 0,C 180,E1 -11562.603,E2 -11562.603} C_VEL
LIN {X 0,Y 391.659,Z 127.11,A -85,B 0,C 180,E1 -11564.412,E2 -11564.412} C_VEL
LIN {X 0,Y 392.566,Z 129.274,A -85,B 0,C 180,E1 -11567.133,E2 -11567.133} C_VEL
LIN {X 0,Y 393.86,Z 132.703,A -85,B 0,C 180,E1 -11569.598,E2 -11569.598} C_VEL
LIN {X 0,Y 395.789,Z 138.125,A -85,B 0,C 180,E1 -11572.318,E2 -11572.318} C_VEL
LIN {X 0,Y 397.848,Z 144.829,A -85,B 0,C 180,E1 -11574.838,E2 -11574.838} C_VEL
LIN {X 0,Y 399.4,Z 150.566,A -85,B 0,C 180,E1 -11576.638,E2 -11576.638} C_VEL
LIN {X 0,Y 399.877,Z 152.521,A -85,B 0,C 180,E1 -11577.13,E2 -11577.13} C_VEL
LIN {X 0,Y 403.272,Z 159.355,A -85,B 0,C 180,E1 -11578.077,E2 -11578.077} C_VEL
LIN {X 0,Y 405.412,Z 164.283,A -85,B 0,C 180,E1 -11578.663,E2 -11578.663} C_VEL
LIN {X 0,Y 407.528,Z 174.998,A -85,B 0,C 180,E1 -11579.46,E2 -11579.46} C_VEL
LIN {X 0,Y 409.843,Z 190.274,A -85,B 0,C 180,E1 -11580.41,E2 -11580.41} C_VEL
LIN {X 0,Y 410.984,Z 203.225,A -85,B 0,C 180,E1 -11581.06,E2 -11581.06} C_VEL
LIN {X 0,Y 405.6,Z 283.345,A -85,B 0,C 180,E1 -11583.293,E2 -11583.293} C_VEL
LIN {X 0,Y 403.2,Z 326.611,A -85,B 0,C 180,E1 -11584.478,E2 -11584.478} C_VEL
LIN {X 0,Y 401.77,Z 343.024,A -85,B 0,C 180,E1 -11585.108,E2 -11585.108} C_VEL
LIN {X 0,Y 400.22,Z 358.386,A -85,B 0,C 180,E1 -11585.904,E2 -11585.904} C_VEL
LIN {X 0,Y 398.603,Z 372.917,A -85,B 0,C 180,E1 -11586.857,E2 -11586.857} C_VEL
LIN {X 0,Y 396.764,Z 390.277,A -85,B 0,C 180,E1 -11588.162,E2 -11588.162} C_VEL
LIN {X 0,Y 395.449,Z 402.632,A -85,B 0,C 180,E1 -11589.315,E2 -11589.315} C_VEL
LIN {X 0,Y 394.113,Z 414.11,A -85,B 0,C 180,E1 -11590.602,E2 -11590.602} C_VEL
LIN {X 0,Y 392.869,Z 424.76,A -85,B 0,C 180,E1 -11592.026,E2 -11592.026} C_VEL
LIN {X 0,Y 391.763,Z 434.599,A -85,B 0,C 180,E1 -11593.588,E2 -11593.588} C_VEL
LIN {X 0,Y 390.645,Z 444.206,A -85,B 0,C 180,E1 -11595.412,E2 -11595.412} C_VEL
LIN {X 0,Y 389.903,Z 451.932,A -85,B 0,C 180,E1 -11597.178,E2 -11597.178} C_VEL
LIN {X 0,Y 389.349,Z 458.789,A -85,B 0,C 180,E1 -11599.075,E2 -11599.075} C_VEL
LIN {X 0,Y 388.947,Z 464.831,A -85,B 0,C 180,E1 -11601.165,E2 -11601.165} C_VEL
LIN {X 0,Y 388.826,Z 468.393,A -85,B 0,C 180,E1 -11602.731,E2 -11602.731} C_VEL
LIN {X 0,Y 388.699,Z 472.009,A -85,B 0,C 180,E1 -11604.813,E2 -11604.813} C_VEL
LIN {X 0,Y 388.652,Z 474.375,A -85,B 0,C 180,E1 -11606.89,E2 -11606.89} C_VEL
LIN {X 0,Y 388.713,Z 475.543,A -85,B 0,C 180,E1 -11608.964,E2 -11608.964} C_VEL
LIN {X 0,Y 388.712,Z 475.52,A -85,B 0,C 180,E1 -11611.036,E2 -11611.036} C_VEL
LIN {X 0,Y 388.653,Z 474.268,A -85,B 0,C 180,E1 -11613.11,E2 -11613.11} C_VEL
LIN {X 0,Y 388.703,Z 471.796,A -85,B 0,C 180,E1 -11615.187,E2 -11615.187} C_VEL
LIN {X 0,Y 388.825,Z 468.054,A -85,B 0,C 180,E1 -11617.269,E2 -11617.269} C_VEL
LIN {X 0,Y 388.979,Z 462.952,A -85,B 0,C 180,E1 -11619.358,E2 -11619.358} C_VEL
LIN {X 0,Y 389.469,Z 456.363,A -85,B 0,C 180,E1 -11621.449,E2 -11621.449} C_VEL
LIN {X 0,Y 389.899,Z 449.328,A -85,B 0,C 180,E1 -11623.256,E2 -11623.256} C_VEL
LIN {X 0,Y 390.837,Z 440.536,A -85,B 0,C 180,E1 -11625.114,E2 -11625.114} C_VEL
LIN {X 0,Y 391.99,Z 430.057,A -85,B 0,C 180,E1 -11626.939,E2 -11626.939} C_VEL
LIN {X 0,Y 393.003,Z 419.539,A -85,B 0,C 180,E1 -11628.466,E2 -11628.466} C_VEL
LIN {X 0,Y 394.349,Z 407.39,A -85,B 0,C 180,E1 -11629.928,E2 -11629.928} C_VEL
LIN {X 0,Y 395.739,Z 394.403,A -85,B 0,C 180,E1 -11631.213,E2 -11631.213} C_VEL
LIN {X 0,Y 397.14,Z 380.004,A -85,B 0,C 180,E1 -11632.363,E2 -11632.363} C_VEL
LIN {X 0,Y 399.22,Z 359.994,A -85,B 0,C 180,E1 -11633.734,E2 -11633.734} C_VEL
LIN {X 0,Y 400.774,Z 344.686,A -85,B 0,C 180,E1 -11634.544,E2 -11634.544} C_VEL
LIN {X 0,Y 402.138,Z 328.874,A -85,B 0,C 180,E1 -11635.179,E2 -11635.179} C_VEL
LIN {X 0,Y 403.497,Z 305.114,A -85,B 0,C 180,E1 -11635.848,E2 -11635.848} C_VEL
LIN {X 0,Y 408.168,Z 228.136,A -85,B 0,C 180,E1 -11637.969,E2 -11637.969} C_VEL
LIN {X 0,Y 410.292,Z 197.144,A -85,B 0,C 180,E1 -11638.876,E2 -11638.876} C_VEL
LIN {X 0,Y 408.914,Z 176.704,A -85,B 0,C 180,E1 -11639.872,E2 -11639.872} C_VEL
LIN {X 0,Y 407.437,Z 162.147,A -85,B 0,C 180,E1 -11640.701,E2 -11640.701} C_VEL
LIN {X 0,Y 403.411,Z 150.658,A -85,B 0,C 180,E1 -11641.874,E2 -11641.874} C_VEL
LIN {X 0,Y 400.45,Z 142.048,A -85,B 0,C 180,E1 -11642.884,E2 -11642.884} C_VEL
LIN {X 0,Y 399.291,Z 137.722,A -85,B 0,C 180,E1 -11643.458,E2 -11643.458} C_VEL
LIN {X 0,Y 398.041,Z 135.405,A -85,B 0,C 180,E1 -11643.917,E2 -11643.917} C_VEL
LIN {X 0,Y 396.38,Z 132.394,A -85,B 0,C 180,E1 -11644.567,E2 -11644.567} C_VEL
LIN {X 0,Y 394.942,Z 130.893,A -85,B 0,C 180,E1 -11645.058,E2 -11645.058} C_VEL
LIN {X 0,Y 393.414,Z 127.72,A -85,B 0,C 180,E1 -11645.794,E2 -11645.794} C_VEL
LIN {X 0,Y 391.036,Z 125.345,A -85,B 0,C 180,E1 -11646.772,E2 -11646.772} C_VEL
LIN {X 0,Y 390.052,Z 122.524,A -85,B 0,C 180,E1 -11647.501,E2 -11647.501} C_VEL
LIN {X 0,Y 390.015,Z 122.527,A -85,B 0,C 180,E1 -11650.815,E2 -11650.815} C_VEL
LIN {X 0,Y 390.043,Z 122.52,A -85,B 0,C 180,E1 -11653.885,E2 -11653.885} C_VEL
LIN {X 0,Y 390.046,Z 122.523,A -85,B 0,C 180,E1 -11656.788,E2 -11656.788} C_VEL
LIN {X 0,Y 390.008,Z 122.527,A -85,B 0,C 180,E1 -11659.555,E2 -11659.555} C_VEL
LIN {X 0,Y 390.039,Z 122.524,A -85,B 0,C 180,E1 -11662.45,E2 -11662.45} C_VEL
LIN {X 0,Y 390.063,Z 122.661,A -85,B 0,C 180,E1 -11663.565,E2 -11663.565} C_VEL
LIN {X 0,Y 391.018,Z 125.305,A -85,B 0,C 180,E1 -11664.51,E2 -11664.51} C_VEL
LIN {X 0,Y 392.815,Z 128.314,A -85,B 0,C 180,E1 -11665.665,E2 -11665.665} C_VEL
LIN {X 0,Y 396.22,Z 132.837,A -85,B 0,C 180,E1 -11666.748,E2 -11666.748} C_VEL
LIN {X 0,Y 399.47,Z 137.531,A -85,B 0,C 180,E1 -11667.698,E2 -11667.698} C_VEL
LIN {X 0,Y 404.304,Z 144.813,A -85,B 0,C 180,E1 -11668.95,E2 -11668.95} C_VEL
LIN {X 0,Y 408.815,Z 152.822,A -85,B 0,C 180,E1 -11670.038,E2 -11670.038} C_VEL
LIN {X 0,Y 412.745,Z 160.761,A -85,B 0,C 180,E1 -11670.935,E2 -11670.935} C_VEL
LIN {X 0,Y 407.396,Z 234.414,A -85,B 0,C 180,E1 -11673.04,E2 -11673.04} C_VEL
LIN {X 0,Y 404.039,Z 292.311,A -85,B 0,C 180,E1 -11674.639,E2 -11674.639} C_VEL
LIN {X 0,Y 402.927,Z 308.825,A -85,B 0,C 180,E1 -11675.316,E2 -11675.316} C_VEL
LIN {X 0,Y 401.667,Z 324.022,A -85,B 0,C 180,E1 -11676.157,E2 -11676.157} C_VEL
LIN {X 0,Y 400.37,Z 338.052,A -85,B 0,C 180,E1 -11677.147,E2 -11677.147} C_VEL
LIN {X 0,Y 398.863,Z 351.351,A -85,B 0,C 180,E1 -11678.283,E2 -11678.283} C_VEL
LIN {X 0,Y 397.302,Z 364.391,A -85,B 0,C 180,E1 -11679.642,E2 -11679.642} C_VEL
LIN {X 0,Y 395.968,Z 374.124,A -85,B 0,C 180,E1 -11680.831,E2 -11680.831} C_VEL
LIN {X 0,Y 394.528,Z 384.787,A -85,B 0,C 180,E1 -11682.372,E2 -11682.372} C_VEL
LIN {X 0,Y 393.239,Z 395.141,A -85,B 0,C 180,E1 -11684.184,E2 -11684.184} C_VEL
LIN {X 0,Y 391.955,Z 403.94,A -85,B 0,C 180,E1 -11686.031,E2 -11686.031} C_VEL
LIN {X 0,Y 391.157,Z 409.992,A -85,B 0,C 180,E1 -11687.549,E2 -11687.549} C_VEL
LIN {X 0,Y 390.533,Z 415.195,A -85,B 0,C 180,E1 -11689.108,E2 -11689.108} C_VEL
LIN {X 0,Y 389.896,Z 420.812,A -85,B 0,C 180,E1 -11691.187,E2 -11691.187} C_VEL
LIN {X 0,Y 389.459,Z 424.548,A -85,B 0,C 180,E1 -11692.982,E2 -11692.982} C_VEL
LIN {X 0,Y 389.075,Z 427.317,A -85,B 0,C 180,E1 -11694.818,E2 -11694.818} C_VEL
LIN {X 0,Y 389.14,Z 428.42,A -85,B 0,C 180,E1 -11695.858,E2 -11695.858} C_VEL
LIN {X 0,Y 388.925,Z 429.727,A -85,B 0,C 180,E1 -11697.929,E2 -11697.929} C_VEL
LIN {X 0,Y 388.795,Z 429.795,A -85,B 0,C 180,E1 -11700,E2 -11700} C_VEL
LIN {X 0,Y 388.883,Z 428.621,A -85,B 0,C 180,E1 -11702.072,E2 -11702.072} C_VEL
LIN {X 0,Y 388.894,Z 426.202,A -85,B 0,C 180,E1 -11704.146,E2 -11704.146} C_VEL
LIN {X 0,Y 389.097,Z 422.47,A -85,B 0,C 180,E1 -11706.222,E2 -11706.222} C_VEL
LIN {X 0,Y 389.34,Z 417.347,A -85,B 0,C 180,E1 -11708.303,E2 -11708.303} C_VEL
LIN {X 0,Y 389.735,Z 410.698,A -85,B 0,C 180,E1 -11710.389,E2 -11710.389} C_VEL
LIN {X 0,Y 390.446,Z 402.323,A -85,B 0,C 180,E1 -11712.475,E2 -11712.475} C_VEL
LIN {X 0,Y 390.93,Z 394.593,A -85,B 0,C 180,E1 -11714.072,E2 -11714.072} C_VEL
LIN {X 0,Y 391.852,Z 384.163,A -85,B 0,C 180,E1 -11715.874,E2 -11715.874} C_VEL
LIN {X 0,Y 392.827,Z 373.321,A -85,B 0,C 180,E1 -11717.438,E2 -11717.438} C_VEL
LIN {X 0,Y 393.869,Z 361.219,A -85,B 0,C 180,E1 -11718.903,E2 -11718.903} C_VEL
LIN {X 0,Y 394.986,Z 348.696,A -85,B 0,C 180,E1 -11720.166,E2 -11720.166} C_VEL
LIN {X 0,Y 395.964,Z 334.694,A -85,B 0,C 180,E1 -11721.338,E2 -11721.338} C_VEL
LIN {X 0,Y 397.005,Z 320.296,A -85,B 0,C 180,E1 -11722.303,E2 -11722.303} C_VEL
LIN {X 0,Y 397.794,Z 305.287,A -85,B 0,C 180,E1 -11723.096,E2 -11723.096} C_VEL
LIN {X 0,Y 398.476,Z 289.582,A -85,B 0,C 180,E1 -11723.71,E2 -11723.71} C_VEL
LIN {X 0,Y 399.027,Z 271.699,A -85,B 0,C 180,E1 -11724.174,E2 -11724.174} C_VEL
LIN {X 0,Y 402.64,Z 152.795,A -85,B 0,C 180,E1 -11726.854,E2 -11726.854} C_VEL
LIN {X 0,Y 396.365,Z 137.467,A -85,B 0,C 180,E1 -11727.607,E2 -11727.607} C_VEL
LIN {X 0,Y 390.156,Z 123.171,A -85,B 0,C 180,E1 -11728.347,E2 -11728.347} C_VEL
LIN {X 0,Y 390.041,Z 122.525,A -85,B 0,C 180,E1 -11728.407,E2 -11728.407} C_VEL
LIN {X 0,Y 390.025,Z 122.53,A -85,B 0,C 180,E1 -11731.505,E2 -11731.505} C_VEL
LIN {X 0,Y 390.083,Z 122.521,A -85,B 0,C 180,E1 -11735.208,E2 -11735.208} C_VEL
LIN {X 0,Y 390.06,Z 122.523,A -85,B 0,C 180,E1 -11739.097,E2 -11739.097} C_VEL
LIN {X 0,Y 390.032,Z 122.523,A -85,B 0,C 180,E1 -11742.372,E2 -11742.372} C_VEL
LIN {X 0,Y 390.043,Z 122.507,A -85,B 0,C 180,E1 -11745.354,E2 -11745.354} C_VEL
LIN {X 0,Y 390.017,Z 122.516,A -85,B 0,C 180,E1 -11748.185,E2 -11748.185} C_VEL
LIN {X 0,Y 390.062,Z 122.524,A -85,B 0,C 180,E1 -11750.904,E2 -11750.904} C_VEL
LIN {X 0,Y 390.072,Z 122.502,A -85,B 0,C 180,E1 -11754.792,E2 -11754.792} C_VEL
LIN {X 0,Y 390.024,Z 122.527,A -85,B 0,C 180,E1 -11758.496,E2 -11758.496} C_VEL
LIN {X 0,Y 390.031,Z 122.52,A -85,B 0,C 180,E1 -11762.063,E2 -11762.063} C_VEL
LIN {X 0,Y 390.045,Z 122.512,A -85,B 0,C 180,E1 -11765.517,E2 -11765.517} C_VEL
LIN {X 0,Y 390.057,Z 122.52,A -85,B 0,C 180,E1 -11768.878,E2 -11768.878} C_VEL
LIN {X 0,Y 390.093,Z 122.519,A -85,B 0,C 180,E1 -11772.165,E2 -11772.165} C_VEL
LIN {X 0,Y 390.094,Z 122.519,A -85,B 0,C 180,E1 -11775.391,E2 -11775.391} C_VEL
LIN {X 0,Y 390.174,Z 122.506,A -85,B 0,C 180,E1 -11777.517,E2 -11777.517} C_VEL
LIN {X 0,Y 390.191,Z 122.508,A -85,B 0,C 180,E1 -11780.671,E2 -11780.671} C_VEL
LIN {X 0,Y 390.276,Z 122.495,A -85,B 0,C 180,E1 -11783.797,E2 -11783.797} C_VEL
LIN {X 0,Y 390.247,Z 122.546,A -85,B 0,C 180,E1 -11784.445,E2 -11784.445} C_VEL
LIN {X 0,Y 394.539,Z 138.233,A -85,B 0,C 180,E1 -11787.322,E2 -11787.322} C_VEL
LIN {X 0,Y 395.832,Z 143.81,A -85,B 0,C 180,E1 -11788.266,E2 -11788.266} C_VEL
LIN {X 0,Y 400.773,Z 156.269,A -85,B 0,C 180,E1 -11788.884,E2 -11788.884} C_VEL
LIN {X 0,Y 404.711,Z 175.249,A -85,B 0,C 180,E1 -11789.547,E2 -11789.547} C_VEL
LIN {X 0,Y 404.16,Z 199.123,A -85,B 0,C 180,E1 -11789.983,E2 -11789.983} C_VEL
LIN {X 0,Y 403.47,Z 204.974,A -85,B 0,C 180,E1 -11790.051,E2 -11790.051} C_VEL
LIN {X 0,Y 397.782,Z 224.009,A -85,B 0,C 180,E1 -11790.039,E2 -11790.039} C_VEL
LIN {X 0,Y 397.081,Z 229.861,A -85,B 0,C 180,E1 -11790.108,E2 -11790.108} C_VEL
LIN {X 0,Y 395.298,Z 310.442,A -85,B 0,C 180,E1 -11791.624,E2 -11791.624} C_VEL
LIN {X 0,Y 394.598,Z 325.85,A -85,B 0,C 180,E1 -11792.106,E2 -11792.106} C_VEL
LIN {X 0,Y 393.674,Z 340.82,A -85,B 0,C 180,E1 -11792.787,E2 -11792.787} C_VEL
LIN {X 0,Y 392.555,Z 354.363,A -85,B 0,C 180,E1 -11793.593,E2 -11793.593} C_VEL
LIN {X 0,Y 391.251,Z 368.196,A -85,B 0,C 180,E1 -11794.636,E2 -11794.636} C_VEL
LIN {X 0,Y 389.853,Z 380.942,A -85,B 0,C 180,E1 -11795.82,E2 -11795.82} C_VEL
LIN {X 0,Y 388.299,Z 393.817,A -85,B 0,C 180,E1 -11797.279,E2 -11797.279} C_VEL
LIN {X 0,Y 386.842,Z 405.495,A -85,B 0,C 180,E1 -11798.883,E2 -11798.883} C_VEL
LIN {X 0,Y 385.582,Z 415.338,A -85,B 0,C 180,E1 -11800.502,E2 -11800.502} C_VEL
LIN {X 0,Y 384.394,Z 424.953,A -85,B 0,C 180,E1 -11802.406,E2 -11802.406} C_VEL
LIN {X 0,Y 383.45,Z 432.754,A -85,B 0,C 180,E1 -11804.271,E2 -11804.271} C_VEL
LIN {X 0,Y 382.799,Z 438.725,A -85,B 0,C 180,E1 -11805.985,E2 -11805.985} C_VEL
LIN {X 0,Y 382.203,Z 444.944,A -85,B 0,C 180,E1 -11808.216,E2 -11808.216} C_VEL
LIN {X 0,Y 381.785,Z 449.678,A -85,B 0,C 180,E1 -11810.472,E2 -11810.472} C_VEL
LIN {X 0,Y 381.524,Z 453.014,A -85,B 0,C 180,E1 -11812.758,E2 -11812.758} C_VEL
LIN {X 0,Y 381.385,Z 454.976,A -85,B 0,C 180,E1 -11815.077,E2 -11815.077} C_VEL
LIN {X 0,Y 381.352,Z 455.548,A -85,B 0,C 180,E1 -11817.434,E2 -11817.434} C_VEL
LIN {X 0,Y 381.43,Z 454.667,A -85,B 0,C 180,E1 -11819.834,E2 -11819.834} C_VEL
LIN {X 0,Y 381.623,Z 452.483,A -85,B 0,C 180,E1 -11822.097,E2 -11822.097} C_VEL
LIN {X 0,Y 381.936,Z 449.433,A -85,B 0,C 180,E1 -11824.101,E2 -11824.101} C_VEL
LIN {X 0,Y 382.307,Z 445.393,A -85,B 0,C 180,E1 -11826.034,E2 -11826.034} C_VEL
LIN {X 0,Y 382.92,Z 439.564,A -85,B 0,C 180,E1 -11828.187,E2 -11828.187} C_VEL
LIN {X 0,Y 383.746,Z 432.654,A -85,B 0,C 180,E1 -11830.209,E2 -11830.209} C_VEL
LIN {X 0,Y 384.829,Z 424.309,A -85,B 0,C 180,E1 -11832.198,E2 -11832.198} C_VEL
LIN {X 0,Y 386.201,Z 414.519,A -85,B 0,C 180,E1 -11834.112,E2 -11834.112} C_VEL
LIN {X 0,Y 387.717,Z 403.315,A -85,B 0,C 180,E1 -11835.912,E2 -11835.912} C_VEL
LIN {X 0,Y 389.21,Z 392.238,A -85,B 0,C 180,E1 -11837.39,E2 -11837.39} C_VEL
LIN {X 0,Y 390.81,Z 379.719,A -85,B 0,C 180,E1 -11838.773,E2 -11838.773} C_VEL
LIN {X 0,Y 392.373,Z 366.136,A -85,B 0,C 180,E1 -11839.999,E2 -11839.999} C_VEL
LIN {X 0,Y 393.784,Z 351.873,A -85,B 0,C 180,E1 -11841.03,E2 -11841.03} C_VEL
LIN {X 0,Y 394.977,Z 337.551,A -85,B 0,C 180,E1 -11841.836,E2 -11841.836} C_VEL
LIN {X 0,Y 395.911,Z 322.483,A -85,B 0,C 180,E1 -11842.466,E2 -11842.466} C_VEL
LIN {X 0,Y 396.574,Z 307.345,A -85,B 0,C 180,E1 -11842.89,E2 -11842.89} C_VEL
LIN {X 0,Y 399.847,Z 171.108,A -85,B 0,C 180,E1 -11845.459,E2 -11845.459} C_VEL
LIN {X 0,Y 398.13,Z 161.903,A -85,B 0,C 180,E1 -11845.797,E2 -11845.797} C_VEL
LIN {X 0,Y 390.548,Z 144.935,A -85,B 0,C 180,E1 -11846.827,E2 -11846.827} C_VEL
LIN {X 0,Y 389.493,Z 142.544,A -85,B 0,C 180,E1 -11846.995,E2 -11846.995} C_VEL
LIN {X 0,Y 384.758,Z 128.592,A -85,B 0,C 180,E1 -11849.239,E2 -11849.239} C_VEL
LIN {X 0,Y 383.001,Z 123.398,A -85,B 0,C 180,E1 -11850.11,E2 -11850.11} C_VEL
LIN {X 0,Y 383.077,Z 123.583,A -85,B 0,C 180,E1 -11851.249,E2 -11851.249} C_VEL
LIN {X 0,Y 384.887,Z 128.22,A -85,B 0,C 180,E1 -11851.488,E2 -11851.488} C_VEL
LIN {X 0,Y 396.126,Z 154.201,A -85,B 0,C 180,E1 -11852.847,E2 -11852.847} C_VEL
LIN {X 0,Y 391.884,Z 286.707,A -85,B 0,C 180,E1 -11855.961,E2 -11855.961} C_VEL
LIN {X 0,Y 391.228,Z 302.493,A -85,B 0,C 180,E1 -11856.544,E2 -11856.544} C_VEL
LIN {X 0,Y 390.411,Z 317.435,A -85,B 0,C 180,E1 -11857.299,E2 -11857.299} C_VEL
LIN {X 0,Y 389.378,Z 332.509,A -85,B 0,C 180,E1 -11858.283,E2 -11858.283} C_VEL
LIN {X 0,Y 388.245,Z 347.001,A -85,B 0,C 180,E1 -11859.468,E2 -11859.468} C_VEL
LIN {X 0,Y 387.152,Z 359.666,A -85,B 0,C 180,E1 -11860.728,E2 -11860.728} C_VEL
LIN {X 0,Y 386.061,Z 372.332,A -85,B 0,C 180,E1 -11862.246,E2 -11862.246} C_VEL
LIN {X 0,Y 385.052,Z 383.435,A -85,B 0,C 180,E1 -11863.838,E2 -11863.838} C_VEL
LIN {X 0,Y 384.072,Z 394.141,A -85,B 0,C 180,E1 -11865.678,E2 -11865.678} C_VEL
LIN {X 0,Y 383.416,Z 403.194,A -85,B 0,C 180,E1 -11867.562,E2 -11867.562} C_VEL
LIN {X 0,Y 382.747,Z 410.591,A -85,B 0,C 180,E1 -11869.419,E2 -11869.419} C_VEL
LIN {X 0,Y 382.304,Z 417.426,A -85,B 0,C 180,E1 -11871.543,E2 -11871.543} C_VEL
LIN {X 0,Y 382.024,Z 422.704,A -85,B 0,C 180,E1 -11873.662,E2 -11873.662} C_VEL
LIN {X 0,Y 381.845,Z 426.576,A -85,B 0,C 180,E1 -11875.778,E2 -11875.778} C_VEL
LIN {X 0,Y 381.83,Z 429.143,A -85,B 0,C 180,E1 -11877.89,E2 -11877.89} C_VEL
LIN {X 0,Y 381.733,Z 430.468,A -85,B 0,C 180,E1 -11880,E2 -11880} C_VEL
LIN {X 0,Y 381.879,Z 430.548,A -85,B 0,C 180,E1 -11882.109,E2 -11882.109} C_VEL
LIN {X 0,Y 382.107,Z 429.389,A -85,B 0,C 180,E1 -11884.219,E2 -11884.219} C_VEL
LIN {X 0,Y 382.299,Z 426.965,A -85,B 0,C 180,E1 -11886.332,E2 -11886.332} C_VEL
LIN {X 0,Y 382.764,Z 423.244,A -85,B 0,C 180,E1 -11888.446,E2 -11888.446} C_VEL
LIN {X 0,Y 383.472,Z 418.148,A -85,B 0,C 180,E1 -11890.56,E2 -11890.56} C_VEL
